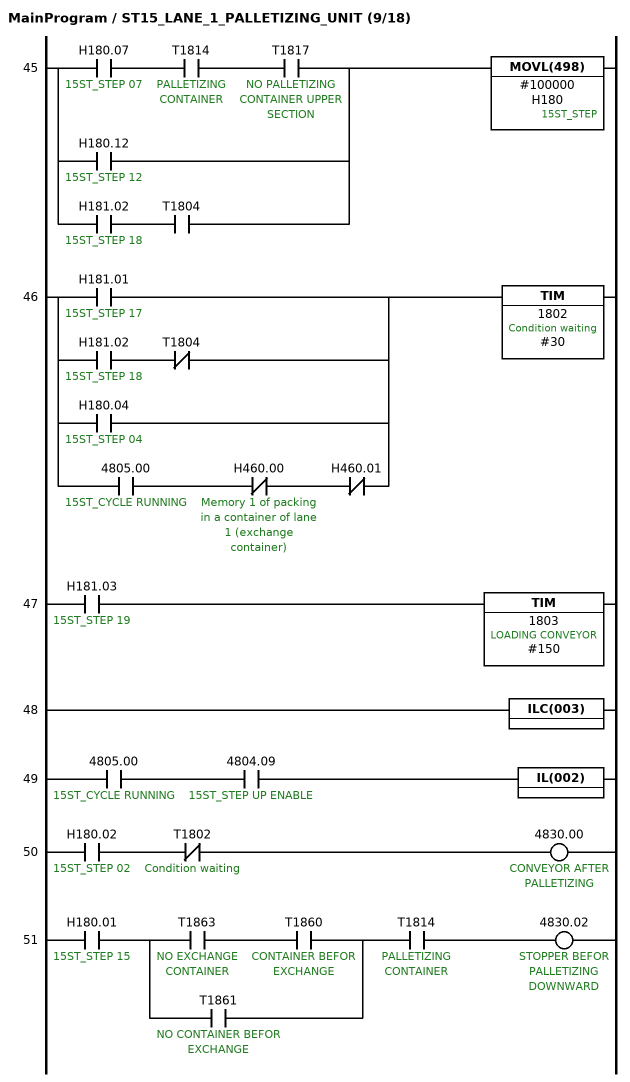
; [picture p624: MainProgram / ST15_LANE_1_PALLETIZING_UNIT, rungs 45-51]
; rung 45
LD H180.07  ; 15ST_STEP 07
AND T1814  ; PALLETIZING CONTAINER
AND T1817  ; NO PALLETIZING CONTAINER UPPER SECTION
OR H180.12  ; 15ST_STEP 12
LD H181.02  ; 15ST_STEP 18
AND T1804
ORLD
MOVL(498) #100000 H180  ; 15ST_STEP
; rung 46
LD H181.01  ; 15ST_STEP 17
LD H181.02  ; 15ST_STEP 18
ANDNOT T1804
ORLD
OR H180.04  ; 15ST_STEP 04
LD 4805.00  ; 15ST_CYCLE RUNNING
ANDNOT H460.00  ; Memory 1 of packing in a container of lane 1 (exchange container)
ANDNOT H460.01
ORLD
TIM 1802 #30  ; Condition waiting
; rung 47
LD H181.03  ; 15ST_STEP 19
TIM 1803 #150  ; LOADING CONVEYOR
; rung 48
ILC(003)
; rung 49
LD 4805.00  ; 15ST_CYCLE RUNNING
AND 4804.09  ; 15ST_STEP UP ENABLE
IL(002)
; rung 50
LD H180.02  ; 15ST_STEP 02
ANDNOT T1802  ; Condition waiting
OUT 4830.00  ; CONVEYOR AFTER PALLETIZING
; rung 51
LD H180.01  ; 15ST_STEP 15
LD T1863  ; NO EXCHANGE CONTAINER
AND T1860  ; CONTAINER BEFOR EXCHANGE
OR T1861  ; NO CONTAINER BEFOR EXCHANGE
ANDLD
AND T1814  ; PALLETIZING CONTAINER
OUT 4830.02  ; STOPPER BEFOR PALLETIZING DOWNWARD

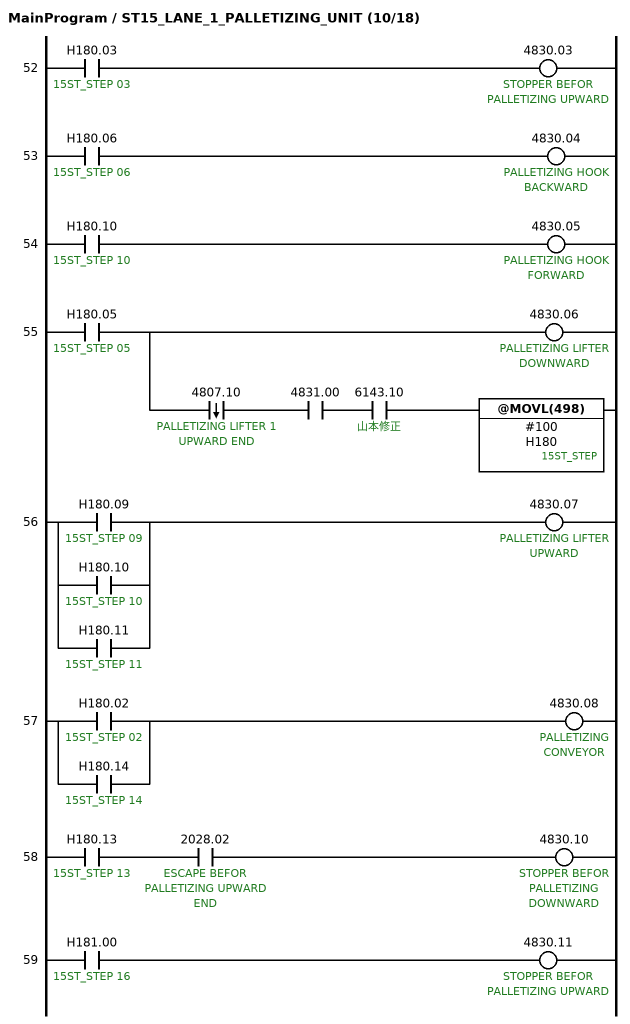
; rung 52
LD H180.03  ; 15ST_STEP 03
OUT 4830.03  ; STOPPER BEFOR PALLETIZING UPWARD
; rung 53
LD H180.06  ; 15ST_STEP 06
OUT 4830.04  ; PALLETIZING HOOK BACKWARD
; rung 54
LD H180.10  ; 15ST_STEP 10
OUT 4830.05  ; PALLETIZING HOOK FORWARD
; rung 55
LD H180.05  ; 15ST_STEP 05
OUT 4830.06  ; PALLETIZING LIFTER DOWNWARD
%AND 4807.10  ; PALLETIZING LIFTER 1 UPWARD END
AND 4831.00
AND 6143.10  ; 山本修正
@MOVL(498) #100 H180  ; 15ST_STEP
; rung 56
LD H180.09  ; 15ST_STEP 09
OR H180.10  ; 15ST_STEP 10
OR H180.11  ; 15ST_STEP 11
OUT 4830.07  ; PALLETIZING LIFTER UPWARD
; rung 57
LD H180.02  ; 15ST_STEP 02
OR H180.14  ; 15ST_STEP 14
OUT 4830.08  ; PALLETIZING CONVEYOR
; rung 58
LD H180.13  ; 15ST_STEP 13
AND 2028.02  ; ESCAPE BEFOR PALLETIZING UPWARD END
OUT 4830.10  ; STOPPER BEFOR PALLETIZING DOWNWARD
; rung 59
LD H181.00  ; 15ST_STEP 16
OUT 4830.11  ; STOPPER BEFOR PALLETIZING UPWARD

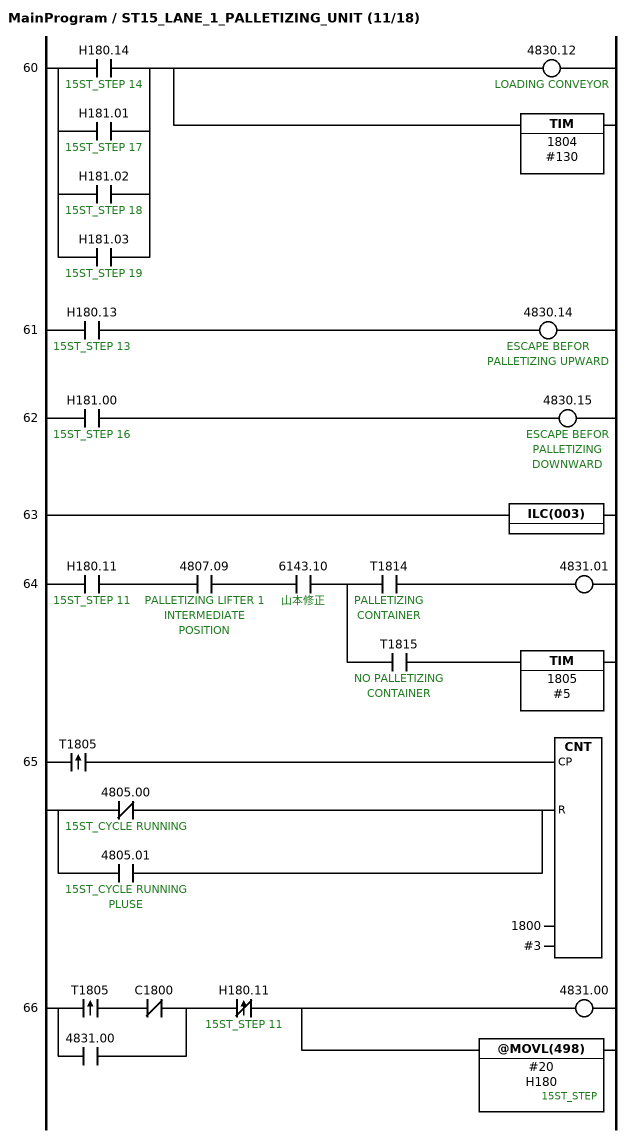
; rung 60
LD H180.14  ; 15ST_STEP 14
OR H181.01  ; 15ST_STEP 17
OR H181.02  ; 15ST_STEP 18
OR H181.03  ; 15ST_STEP 19
OUT 4830.12  ; LOADING CONVEYOR
TIM 1804 #130
; rung 61
LD H180.13  ; 15ST_STEP 13
OUT 4830.14  ; ESCAPE BEFOR PALLETIZING UPWARD
; rung 62
LD H181.00  ; 15ST_STEP 16
OUT 4830.15  ; ESCAPE BEFOR PALLETIZING DOWNWARD
; rung 63
ILC(003)
; rung 64
LD H180.11  ; 15ST_STEP 11
AND 4807.09  ; PALLETIZING LIFTER 1 INTERMEDIATE POSITION
AND 6143.10  ; 山本修正
OUT TR0
AND T1814  ; PALLETIZING CONTAINER
OUT 4831.01
LD TR0
AND T1815  ; NO PALLETIZING CONTAINER
TIM 1805 #5
; rung 65
@LD T1805
LDNOT 4805.00  ; 15ST_CYCLE RUNNING
OR 4805.01  ; 15ST_CYCLE RUNNING PLUSE
CNT 1800 #3
; rung 66
@LD T1805
ANDNOT C1800
OR 4831.00
@ANDNOT H180.11  ; 15ST_STEP 11
OUT 4831.00
@MOVL(498) #20 H180  ; 15ST_STEP

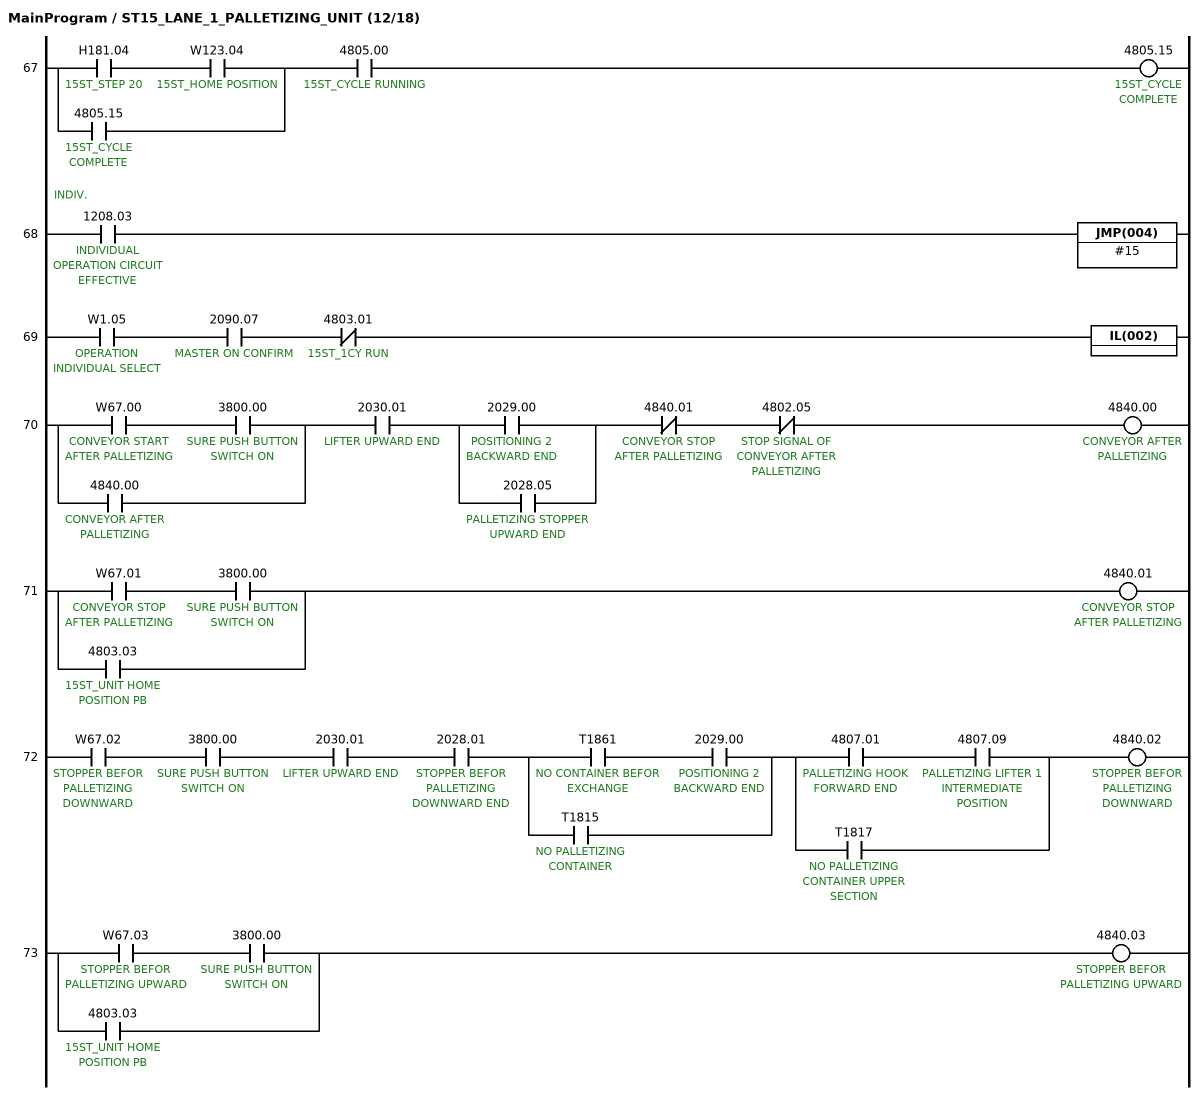
; rung 67
LD H181.04  ; 15ST_STEP 20
AND W123.04  ; 15ST_HOME POSITION
OR 4805.15  ; 15ST_CYCLE COMPLETE
AND 4805.00  ; 15ST_CYCLE RUNNING
OUT 4805.15  ; 15ST_CYCLE COMPLETE
; rung 68: INDIV.
LD 1208.03  ; INDIVIDUAL OPERATION CIRCUIT EFFECTIVE
JMP(004) #15
; rung 69
LD W1.05  ; OPERATION INDIVIDUAL SELECT
AND 2090.07  ; MASTER ON CONFIRM
ANDNOT 4803.01  ; 15ST_1CY RUN
IL(002)
; rung 70
LD W67.00  ; CONVEYOR START AFTER PALLETIZING
AND 3800.00  ; SURE PUSH BUTTON SWITCH ON
OR 4840.00  ; CONVEYOR AFTER PALLETIZING
AND 2030.01  ; LIFTER UPWARD END
LD 2029.00  ; POSITIONING 2 BACKWARD END
OR 2028.05  ; PALLETIZING STOPPER UPWARD END
ANDLD
ANDNOT 4840.01  ; CONVEYOR STOP AFTER PALLETIZING
ANDNOT 4802.05  ; STOP SIGNAL OF CONVEYOR AFTER PALLETIZING
OUT 4840.00  ; CONVEYOR AFTER PALLETIZING
; rung 71
LD W67.01  ; CONVEYOR STOP AFTER PALLETIZING
AND 3800.00  ; SURE PUSH BUTTON SWITCH ON
OR 4803.03  ; 15ST_UNIT HOME POSITION PB
OUT 4840.01  ; CONVEYOR STOP AFTER PALLETIZING
; rung 72
LD W67.02  ; STOPPER BEFOR PALLETIZING DOWNWARD
AND 3800.00  ; SURE PUSH BUTTON SWITCH ON
AND 2030.01  ; LIFTER UPWARD END
AND 2028.01  ; STOPPER BEFOR PALLETIZING DOWNWARD END
LD T1861  ; NO CONTAINER BEFOR EXCHANGE
AND 2029.00  ; POSITIONING 2 BACKWARD END
OR T1815  ; NO PALLETIZING CONTAINER
ANDLD
LD 4807.01  ; PALLETIZING HOOK FORWARD END
AND 4807.09  ; PALLETIZING LIFTER 1 INTERMEDIATE POSITION
OR T1817  ; NO PALLETIZING CONTAINER UPPER SECTION
ANDLD
OUT 4840.02  ; STOPPER BEFOR PALLETIZING DOWNWARD
; rung 73
LD W67.03  ; STOPPER BEFOR PALLETIZING UPWARD
AND 3800.00  ; SURE PUSH BUTTON SWITCH ON
OR 4803.03  ; 15ST_UNIT HOME POSITION PB
OUT 4840.03  ; STOPPER BEFOR PALLETIZING UPWARD

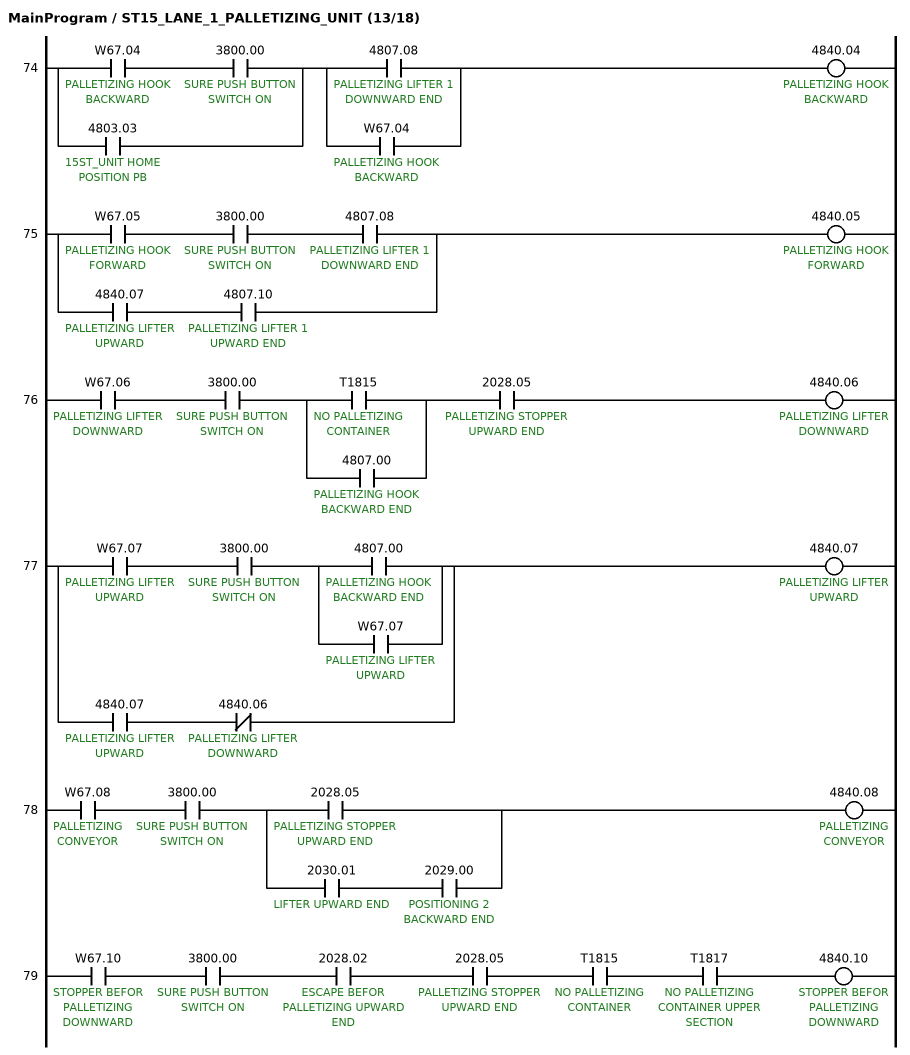
; rung 74
LD W67.04  ; PALLETIZING HOOK BACKWARD
AND 3800.00  ; SURE PUSH BUTTON SWITCH ON
OR 4803.03  ; 15ST_UNIT HOME POSITION PB
LD 4807.08  ; PALLETIZING LIFTER 1 DOWNWARD END
OR W67.04  ; PALLETIZING HOOK BACKWARD
ANDLD
OUT 4840.04  ; PALLETIZING HOOK BACKWARD
; rung 75
LD W67.05  ; PALLETIZING HOOK FORWARD
AND 3800.00  ; SURE PUSH BUTTON SWITCH ON
AND 4807.08  ; PALLETIZING LIFTER 1 DOWNWARD END
LD 4840.07  ; PALLETIZING LIFTER UPWARD
AND 4807.10  ; PALLETIZING LIFTER 1 UPWARD END
ORLD
OUT 4840.05  ; PALLETIZING HOOK FORWARD
; rung 76
LD W67.06  ; PALLETIZING LIFTER DOWNWARD
AND 3800.00  ; SURE PUSH BUTTON SWITCH ON
LD T1815  ; NO PALLETIZING CONTAINER
OR 4807.00  ; PALLETIZING HOOK BACKWARD END
ANDLD
AND 2028.05  ; PALLETIZING STOPPER UPWARD END
OUT 4840.06  ; PALLETIZING LIFTER DOWNWARD
; rung 77
LD W67.07  ; PALLETIZING LIFTER UPWARD
AND 3800.00  ; SURE PUSH BUTTON SWITCH ON
LD 4807.00  ; PALLETIZING HOOK BACKWARD END
OR W67.07  ; PALLETIZING LIFTER UPWARD
ANDLD
LD 4840.07  ; PALLETIZING LIFTER UPWARD
ANDNOT 4840.06  ; PALLETIZING LIFTER DOWNWARD
ORLD
OUT 4840.07  ; PALLETIZING LIFTER UPWARD
; rung 78
LD W67.08  ; PALLETIZING CONVEYOR
AND 3800.00  ; SURE PUSH BUTTON SWITCH ON
LD 2028.05  ; PALLETIZING STOPPER UPWARD END
LD 2030.01  ; LIFTER UPWARD END
AND 2029.00  ; POSITIONING 2 BACKWARD END
ORLD
ANDLD
OUT 4840.08  ; PALLETIZING CONVEYOR
; rung 79
LD W67.10  ; STOPPER BEFOR PALLETIZING DOWNWARD
AND 3800.00  ; SURE PUSH BUTTON SWITCH ON
AND 2028.02  ; ESCAPE BEFOR PALLETIZING UPWARD END
AND 2028.05  ; PALLETIZING STOPPER UPWARD END
AND T1815  ; NO PALLETIZING CONTAINER
AND T1817  ; NO PALLETIZING CONTAINER UPPER SECTION
OUT 4840.10  ; STOPPER BEFOR PALLETIZING DOWNWARD

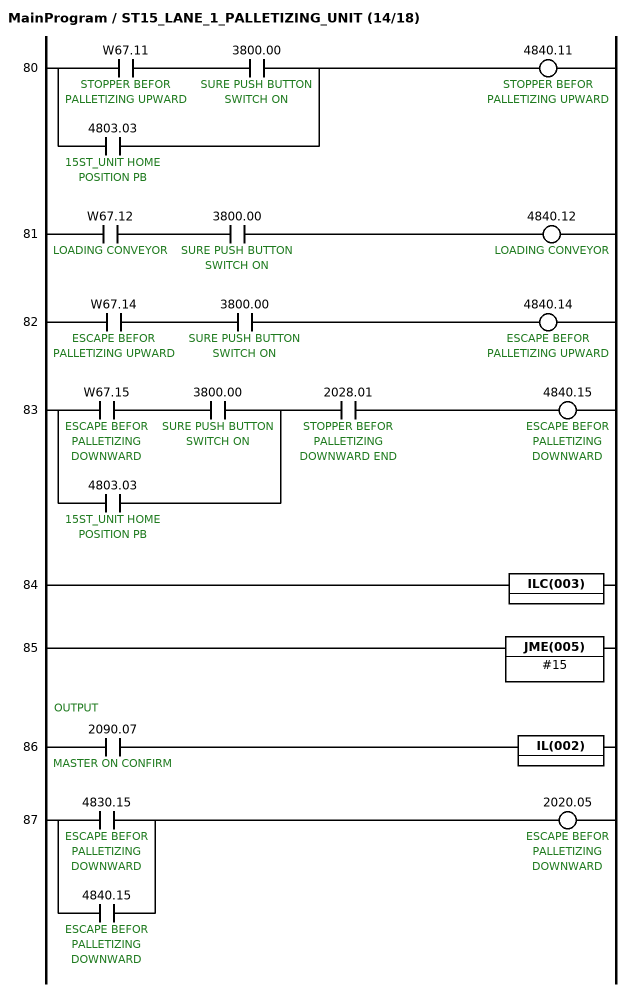
; rung 80
LD W67.11  ; STOPPER BEFOR PALLETIZING UPWARD
AND 3800.00  ; SURE PUSH BUTTON SWITCH ON
OR 4803.03  ; 15ST_UNIT HOME POSITION PB
OUT 4840.11  ; STOPPER BEFOR PALLETIZING UPWARD
; rung 81
LD W67.12  ; LOADING CONVEYOR
AND 3800.00  ; SURE PUSH BUTTON SWITCH ON
OUT 4840.12  ; LOADING CONVEYOR
; rung 82
LD W67.14  ; ESCAPE BEFOR PALLETIZING UPWARD
AND 3800.00  ; SURE PUSH BUTTON SWITCH ON
OUT 4840.14  ; ESCAPE BEFOR PALLETIZING UPWARD
; rung 83
LD W67.15  ; ESCAPE BEFOR PALLETIZING DOWNWARD
AND 3800.00  ; SURE PUSH BUTTON SWITCH ON
OR 4803.03  ; 15ST_UNIT HOME POSITION PB
AND 2028.01  ; STOPPER BEFOR PALLETIZING DOWNWARD END
OUT 4840.15  ; ESCAPE BEFOR PALLETIZING DOWNWARD
; rung 84
ILC(003)
; rung 85
JME(005) #15
; rung 86: OUTPUT
LD 2090.07  ; MASTER ON CONFIRM
IL(002)
; rung 87
LD 4830.15  ; ESCAPE BEFOR PALLETIZING DOWNWARD
OR 4840.15  ; ESCAPE BEFOR PALLETIZING DOWNWARD
OUT 2020.05  ; ESCAPE BEFOR PALLETIZING DOWNWARD

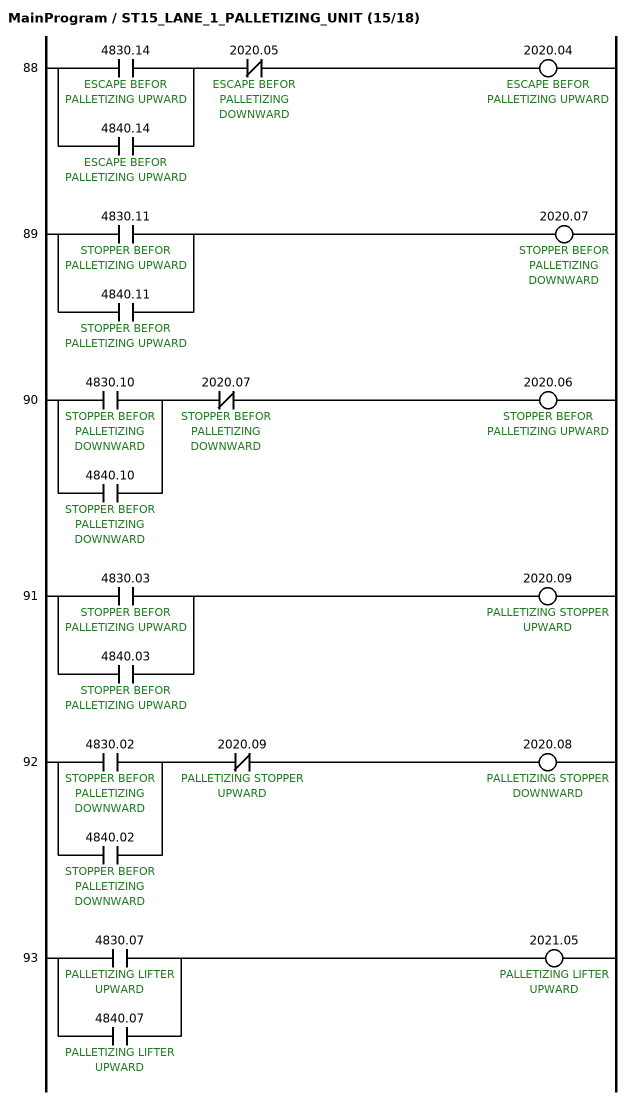
; rung 88
LD 4830.14  ; ESCAPE BEFOR PALLETIZING UPWARD
OR 4840.14  ; ESCAPE BEFOR PALLETIZING UPWARD
ANDNOT 2020.05  ; ESCAPE BEFOR PALLETIZING DOWNWARD
OUT 2020.04  ; ESCAPE BEFOR PALLETIZING UPWARD
; rung 89
LD 4830.11  ; STOPPER BEFOR PALLETIZING UPWARD
OR 4840.11  ; STOPPER BEFOR PALLETIZING UPWARD
OUT 2020.07  ; STOPPER BEFOR PALLETIZING DOWNWARD
; rung 90
LD 4830.10  ; STOPPER BEFOR PALLETIZING DOWNWARD
OR 4840.10  ; STOPPER BEFOR PALLETIZING DOWNWARD
ANDNOT 2020.07  ; STOPPER BEFOR PALLETIZING DOWNWARD
OUT 2020.06  ; STOPPER BEFOR PALLETIZING UPWARD
; rung 91
LD 4830.03  ; STOPPER BEFOR PALLETIZING UPWARD
OR 4840.03  ; STOPPER BEFOR PALLETIZING UPWARD
OUT 2020.09  ; PALLETIZING STOPPER UPWARD
; rung 92
LD 4830.02  ; STOPPER BEFOR PALLETIZING DOWNWARD
OR 4840.02  ; STOPPER BEFOR PALLETIZING DOWNWARD
ANDNOT 2020.09  ; PALLETIZING STOPPER UPWARD
OUT 2020.08  ; PALLETIZING STOPPER DOWNWARD
; rung 93
LD 4830.07  ; PALLETIZING LIFTER UPWARD
OR 4840.07  ; PALLETIZING LIFTER UPWARD
OUT 2021.05  ; PALLETIZING LIFTER UPWARD

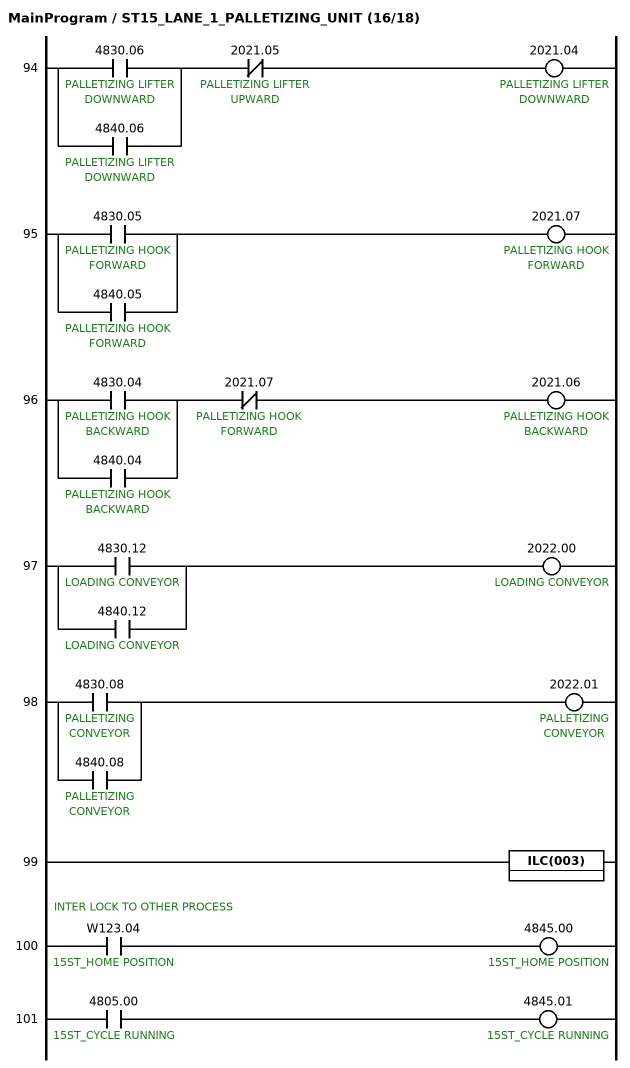
; rung 94
LD 4830.06  ; PALLETIZING LIFTER DOWNWARD
OR 4840.06  ; PALLETIZING LIFTER DOWNWARD
ANDNOT 2021.05  ; PALLETIZING LIFTER UPWARD
OUT 2021.04  ; PALLETIZING LIFTER DOWNWARD
; rung 95
LD 4830.05  ; PALLETIZING HOOK FORWARD
OR 4840.05  ; PALLETIZING HOOK FORWARD
OUT 2021.07  ; PALLETIZING HOOK FORWARD
; rung 96
LD 4830.04  ; PALLETIZING HOOK BACKWARD
OR 4840.04  ; PALLETIZING HOOK BACKWARD
ANDNOT 2021.07  ; PALLETIZING HOOK FORWARD
OUT 2021.06  ; PALLETIZING HOOK BACKWARD
; rung 97
LD 4830.12  ; LOADING CONVEYOR
OR 4840.12  ; LOADING CONVEYOR
OUT 2022.00  ; LOADING CONVEYOR
; rung 98
LD 4830.08  ; PALLETIZING CONVEYOR
OR 4840.08  ; PALLETIZING CONVEYOR
OUT 2022.01  ; PALLETIZING CONVEYOR
; rung 99
ILC(003)
; rung 100: INTER LOCK TO OTHER PROCESS
LD W123.04  ; 15ST_HOME POSITION
OUT 4845.00  ; 15ST_HOME POSITION
; rung 101
LD 4805.00  ; 15ST_CYCLE RUNNING
OUT 4845.01  ; 15ST_CYCLE RUNNING

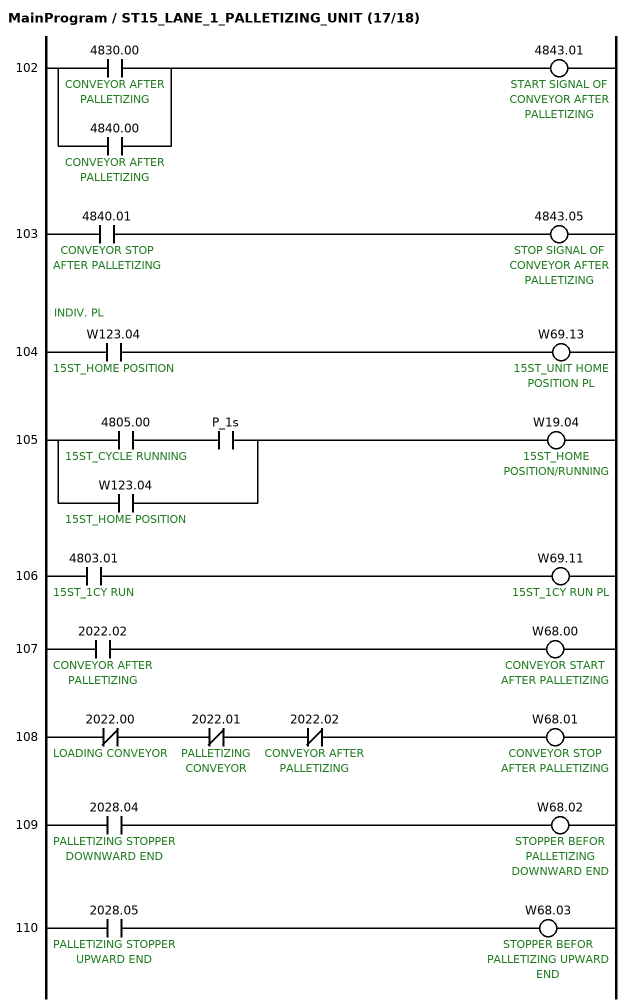
; rung 102
LD 4830.00  ; CONVEYOR AFTER PALLETIZING
OR 4840.00  ; CONVEYOR AFTER PALLETIZING
OUT 4843.01  ; START SIGNAL OF CONVEYOR AFTER PALLETIZING
; rung 103
LD 4840.01  ; CONVEYOR STOP AFTER PALLETIZING
OUT 4843.05  ; STOP SIGNAL OF CONVEYOR AFTER PALLETIZING
; rung 104: INDIV. PL
LD W123.04  ; 15ST_HOME POSITION
OUT W69.13  ; 15ST_UNIT HOME POSITION PL
; rung 105
LD 4805.00  ; 15ST_CYCLE RUNNING
AND P_1s
OR W123.04  ; 15ST_HOME POSITION
OUT W19.04  ; 15ST_HOME POSITION/RUNNING
; rung 106
LD 4803.01  ; 15ST_1CY RUN
OUT W69.11  ; 15ST_1CY RUN PL
; rung 107
LD 2022.02  ; CONVEYOR AFTER PALLETIZING
OUT W68.00  ; CONVEYOR START AFTER PALLETIZING
; rung 108
LDNOT 2022.00  ; LOADING CONVEYOR
ANDNOT 2022.01  ; PALLETIZING CONVEYOR
ANDNOT 2022.02  ; CONVEYOR AFTER PALLETIZING
OUT W68.01  ; CONVEYOR STOP AFTER PALLETIZING
; rung 109
LD 2028.04  ; PALLETIZING STOPPER DOWNWARD END
OUT W68.02  ; STOPPER BEFOR PALLETIZING DOWNWARD END
; rung 110
LD 2028.05  ; PALLETIZING STOPPER UPWARD END
OUT W68.03  ; STOPPER BEFOR PALLETIZING UPWARD END

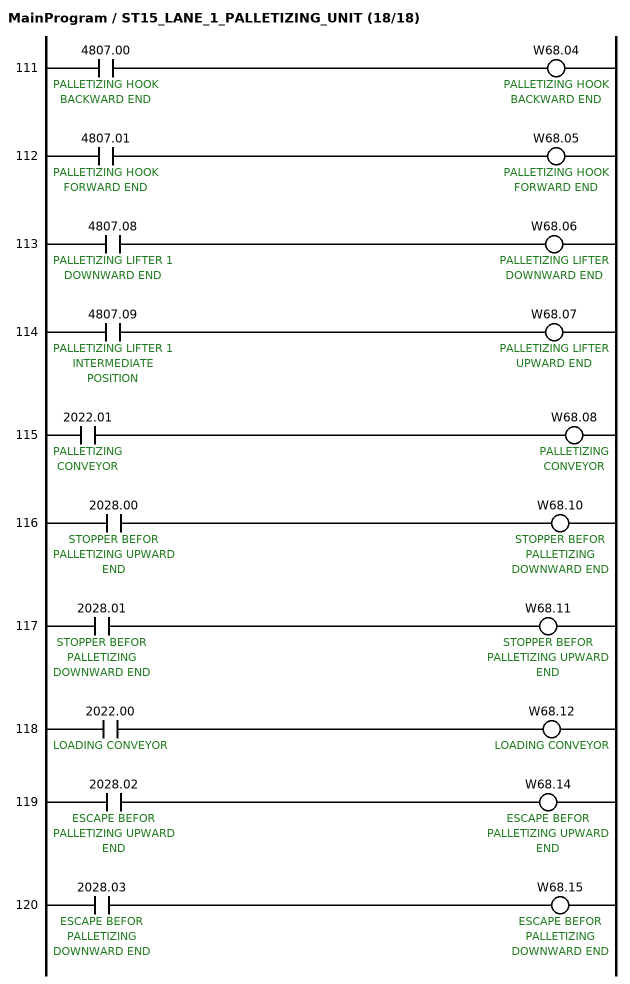
; rung 111
LD 4807.00  ; PALLETIZING HOOK BACKWARD END
OUT W68.04  ; PALLETIZING HOOK BACKWARD END
; rung 112
LD 4807.01  ; PALLETIZING HOOK FORWARD END
OUT W68.05  ; PALLETIZING HOOK FORWARD END
; rung 113
LD 4807.08  ; PALLETIZING LIFTER 1 DOWNWARD END
OUT W68.06  ; PALLETIZING LIFTER DOWNWARD END
; rung 114
LD 4807.09  ; PALLETIZING LIFTER 1 INTERMEDIATE POSITION
OUT W68.07  ; PALLETIZING LIFTER UPWARD END
; rung 115
LD 2022.01  ; PALLETIZING CONVEYOR
OUT W68.08  ; PALLETIZING CONVEYOR
; rung 116
LD 2028.00  ; STOPPER BEFOR PALLETIZING UPWARD END
OUT W68.10  ; STOPPER BEFOR PALLETIZING DOWNWARD END
; rung 117
LD 2028.01  ; STOPPER BEFOR PALLETIZING DOWNWARD END
OUT W68.11  ; STOPPER BEFOR PALLETIZING UPWARD END
; rung 118
LD 2022.00  ; LOADING CONVEYOR
OUT W68.12  ; LOADING CONVEYOR
; rung 119
LD 2028.02  ; ESCAPE BEFOR PALLETIZING UPWARD END
OUT W68.14  ; ESCAPE BEFOR PALLETIZING UPWARD END
; rung 120
LD 2028.03  ; ESCAPE BEFOR PALLETIZING DOWNWARD END
OUT W68.15  ; ESCAPE BEFOR PALLETIZING DOWNWARD END
; rung 121: CONDITION PL

### Section ST16_LANE_1_SUPPLYING_UNIT

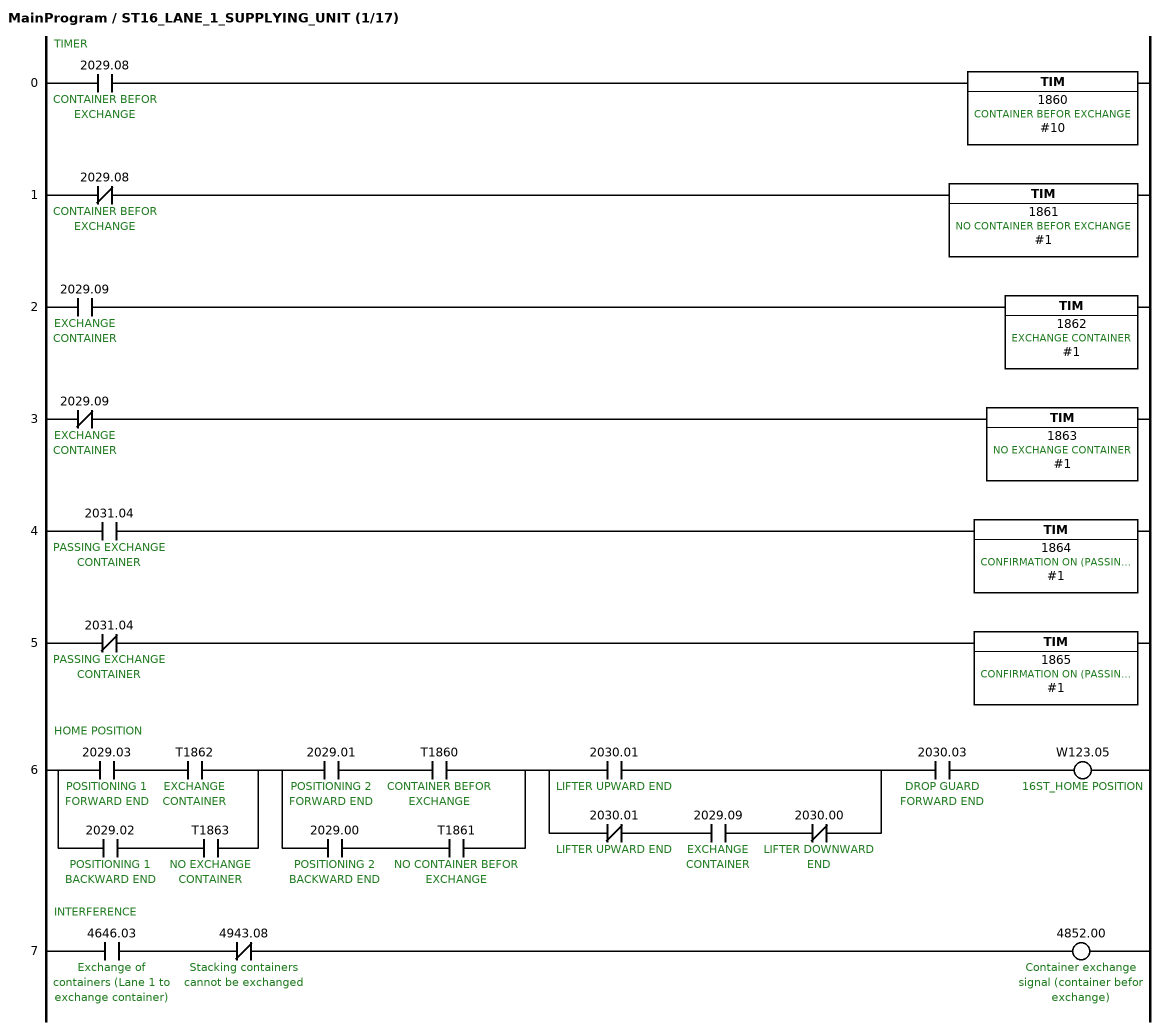
; rung 0: TIMER
LD 2029.08  ; CONTAINER BEFOR EXCHANGE
TIM 1860 #10  ; CONTAINER BEFOR EXCHANGE
; rung 1
LDNOT 2029.08  ; CONTAINER BEFOR EXCHANGE
TIM 1861 #1  ; NO CONTAINER BEFOR EXCHANGE
; rung 2
LD 2029.09  ; EXCHANGE CONTAINER
TIM 1862 #1  ; EXCHANGE CONTAINER
; rung 3
LDNOT 2029.09  ; EXCHANGE CONTAINER
TIM 1863 #1  ; NO EXCHANGE CONTAINER
; rung 4
LD 2031.04  ; PASSING EXCHANGE CONTAINER
TIM 1864 #1  ; CONFIRMATION ON (PASSING EXCHANGE CONTAINER)
; rung 5
LDNOT 2031.04  ; PASSING EXCHANGE CONTAINER
TIM 1865 #1  ; CONFIRMATION ON (PASSING EXCHANGE CONTAINER)
; rung 6: HOME POSITION
LD 2029.03  ; POSITIONING 1 FORWARD END
AND T1862  ; EXCHANGE CONTAINER
LD 2029.02  ; POSITIONING 1 BACKWARD END
AND T1863  ; NO EXCHANGE CONTAINER
ORLD
LD 2029.01  ; POSITIONING 2 FORWARD END
AND T1860  ; CONTAINER BEFOR EXCHANGE
LD 2029.00  ; POSITIONING 2 BACKWARD END
AND T1861  ; NO CONTAINER BEFOR EXCHANGE
ORLD
ANDLD
LD 2030.01  ; LIFTER UPWARD END
LDNOT 2030.01  ; LIFTER UPWARD END
AND 2029.09  ; EXCHANGE CONTAINER
ANDNOT 2030.00  ; LIFTER DOWNWARD END
ORLD
ANDLD
AND 2030.03  ; DROP GUARD FORWARD END
OUT W123.05  ; 16ST_HOME POSITION
; rung 7: INTERFERENCE
LD 4646.03  ; Exchange of containers (Lane 1 to exchange container)
ANDNOT 4943.08  ; Stacking containers cannot be exchanged
OUT 4852.00  ; Container exchange signal (container befor exchange)

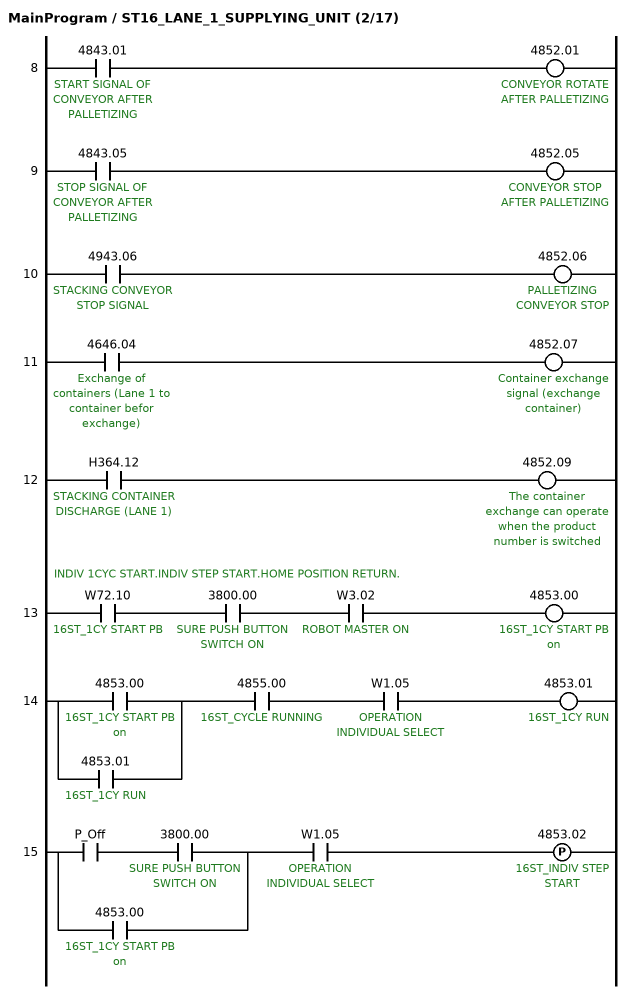
; rung 8
LD 4843.01  ; START SIGNAL OF CONVEYOR AFTER PALLETIZING
OUT 4852.01  ; CONVEYOR ROTATE AFTER PALLETIZING
; rung 9
LD 4843.05  ; STOP SIGNAL OF CONVEYOR AFTER PALLETIZING
OUT 4852.05  ; CONVEYOR STOP AFTER PALLETIZING
; rung 10
LD 4943.06  ; STACKING CONVEYOR STOP SIGNAL
OUT 4852.06  ; PALLETIZING CONVEYOR STOP
; rung 11
LD 4646.04  ; Exchange of containers (Lane 1 to container befor exchange)
OUT 4852.07  ; Container exchange signal (exchange container)
; rung 12
LD H364.12  ; STACKING CONTAINER DISCHARGE (LANE 1)
OUT 4852.09  ; The container exchange can operate when the product number is switched
; rung 13: INDIV 1CYC START.INDIV STEP START.HOME POSITION RETURN.
LD W72.10  ; 16ST_1CY START PB
AND 3800.00  ; SURE PUSH BUTTON SWITCH ON
AND W3.02  ; ROBOT MASTER ON
OUT 4853.00  ; 16ST_1CY START PB on
; rung 14
LD 4853.00  ; 16ST_1CY START PB on
OR 4853.01  ; 16ST_1CY RUN
AND 4855.00  ; 16ST_CYCLE RUNNING
AND W1.05  ; OPERATION INDIVIDUAL SELECT
OUT 4853.01  ; 16ST_1CY RUN
; rung 15
LD P_Off
AND 3800.00  ; SURE PUSH BUTTON SWITCH ON
OR 4853.00  ; 16ST_1CY START PB on
AND W1.05  ; OPERATION INDIVIDUAL SELECT
DIFU(013) 4853.02  ; 16ST_INDIV STEP START

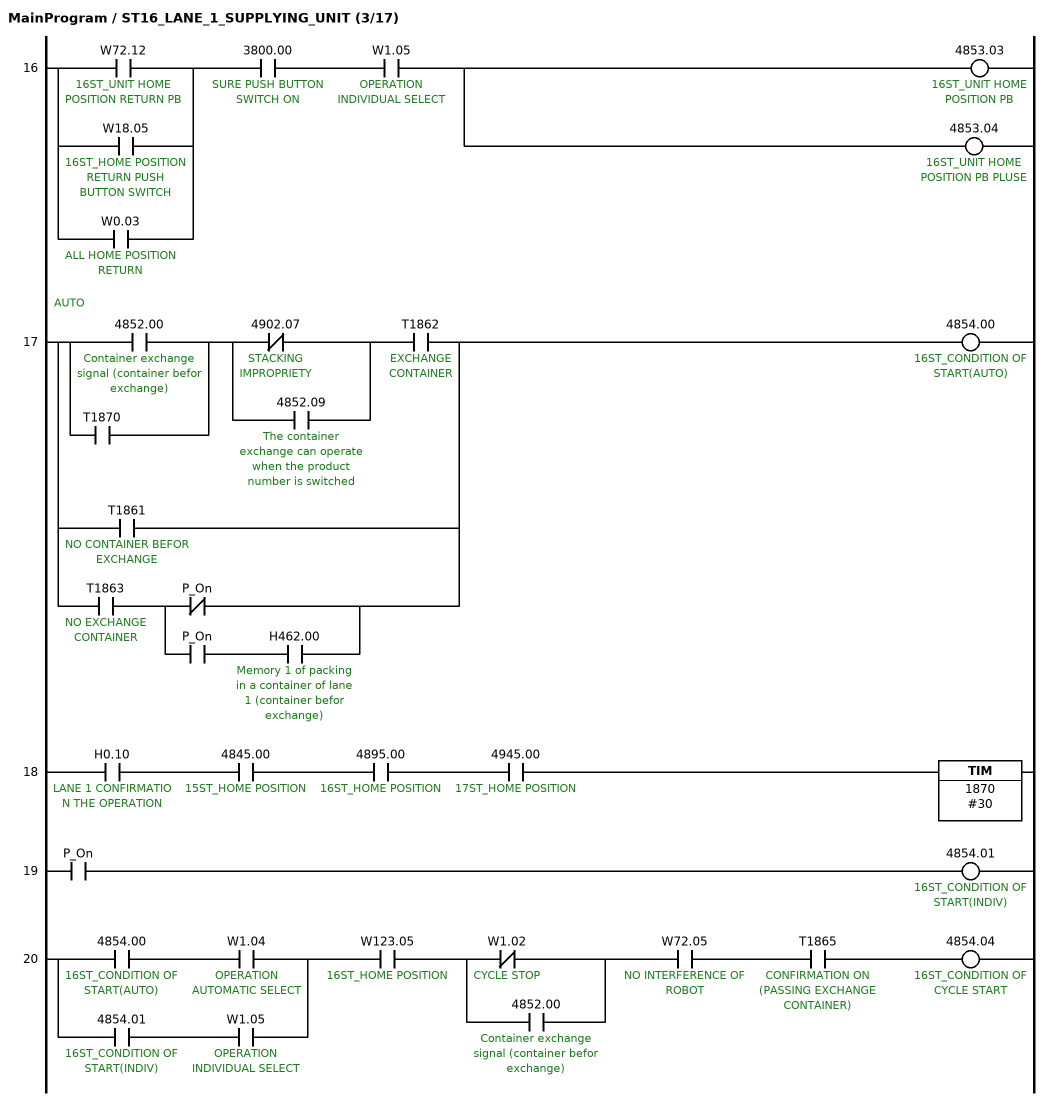
; rung 16
LD W72.12  ; 16ST_UNIT HOME POSITION RETURN PB
OR W18.05  ; 16ST_HOME POSITION RETURN PUSH BUTTON SWITCH
OR W0.03  ; ALL HOME POSITION RETURN
AND 3800.00  ; SURE PUSH BUTTON SWITCH ON
AND W1.05  ; OPERATION INDIVIDUAL SELECT
OUT 4853.03  ; 16ST_UNIT HOME POSITION PB
OUT 4853.04  ; 16ST_UNIT HOME POSITION PB PLUSE
; rung 17: AUTO
LD 4852.00  ; Container exchange signal (container befor exchange)
OR T1870
LDNOT 4902.07  ; STACKING IMPROPRIETY
OR 4852.09  ; The container exchange can operate when the product number is switched
ANDLD
AND T1862  ; EXCHANGE CONTAINER
OR T1861  ; NO CONTAINER BEFOR EXCHANGE
LD T1863  ; NO EXCHANGE CONTAINER
LDNOT P_On
LD P_On
AND H462.00  ; Memory 1 of packing in a container of lane 1 (container befor exchange)
ORLD
ANDLD
ORLD
OUT 4854.00  ; 16ST_CONDITION OF START(AUTO)
; rung 18
LD H0.10  ; LANE 1 CONFIRMATION THE OPERATION
AND 4845.00  ; 15ST_HOME POSITION
AND 4895.00  ; 16ST_HOME POSITION
AND 4945.00  ; 17ST_HOME POSITION
TIM 1870 #30
; rung 19
LD P_On
OUT 4854.01  ; 16ST_CONDITION OF START(INDIV)
; rung 20
LD 4854.00  ; 16ST_CONDITION OF START(AUTO)
AND W1.04  ; OPERATION AUTOMATIC SELECT
LD 4854.01  ; 16ST_CONDITION OF START(INDIV)
AND W1.05  ; OPERATION INDIVIDUAL SELECT
ORLD
AND W123.05  ; 16ST_HOME POSITION
LDNOT W1.02  ; CYCLE STOP
OR 4852.00  ; Container exchange signal (container befor exchange)
ANDLD
AND W72.05  ; NO INTERFERENCE OF ROBOT
AND T1865  ; CONFIRMATION ON (PASSING EXCHANGE CONTAINER)
OUT 4854.04  ; 16ST_CONDITION OF CYCLE START

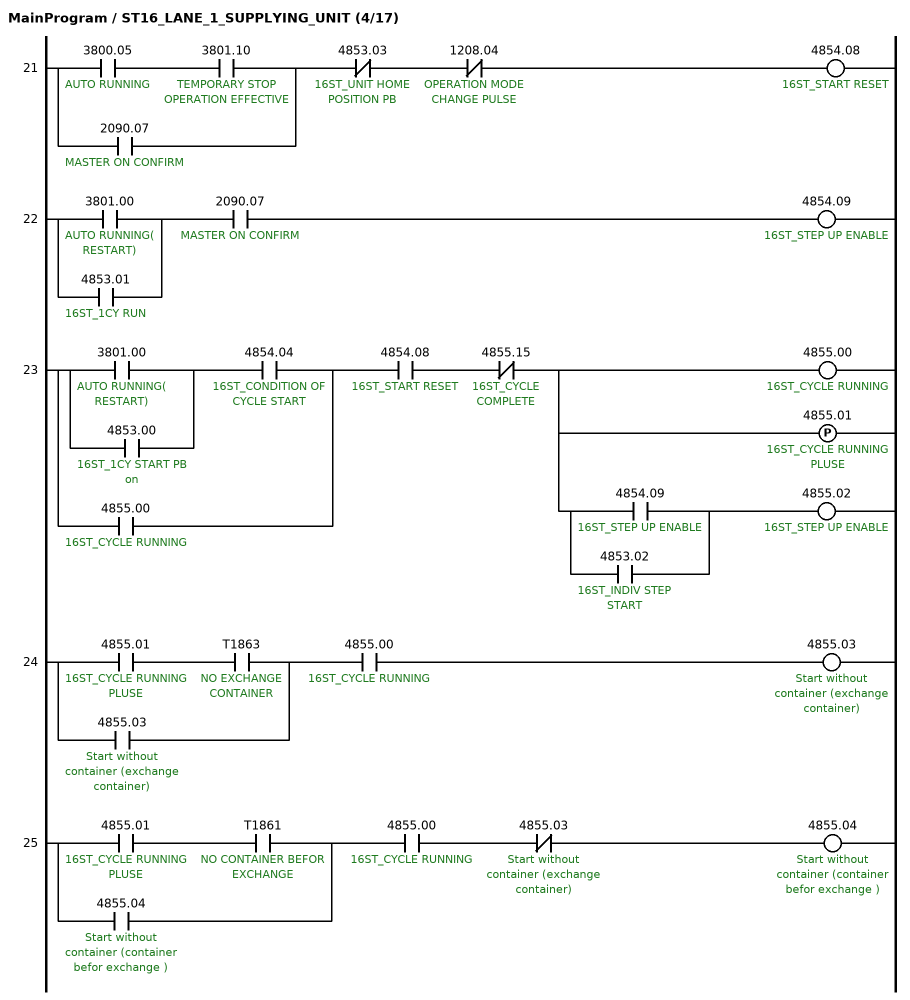
; rung 21
LD 3800.05  ; AUTO RUNNING
AND 3801.10  ; TEMPORARY STOP OPERATION EFFECTIVE
OR 2090.07  ; MASTER ON CONFIRM
ANDNOT 4853.03  ; 16ST_UNIT HOME POSITION PB
ANDNOT 1208.04  ; OPERATION MODE CHANGE PULSE
OUT 4854.08  ; 16ST_START RESET
; rung 22
LD 3801.00  ; AUTO RUNNING(RESTART)
OR 4853.01  ; 16ST_1CY RUN
AND 2090.07  ; MASTER ON CONFIRM
OUT 4854.09  ; 16ST_STEP UP ENABLE
; rung 23
LD 3801.00  ; AUTO RUNNING(RESTART)
OR 4853.00  ; 16ST_1CY START PB on
AND 4854.04  ; 16ST_CONDITION OF CYCLE START
OR 4855.00  ; 16ST_CYCLE RUNNING
AND 4854.08  ; 16ST_START RESET
ANDNOT 4855.15  ; 16ST_CYCLE COMPLETE
OUT 4855.00  ; 16ST_CYCLE RUNNING
DIFU(013) 4855.01  ; 16ST_CYCLE RUNNING PLUSE
LD 4854.09  ; 16ST_STEP UP ENABLE
OR 4853.02  ; 16ST_INDIV STEP START
ANDLD
OUT 4855.02  ; 16ST_STEP UP ENABLE
; rung 24
LD 4855.01  ; 16ST_CYCLE RUNNING PLUSE
AND T1863  ; NO EXCHANGE CONTAINER
OR 4855.03  ; Start without container (exchange container)
AND 4855.00  ; 16ST_CYCLE RUNNING
OUT 4855.03  ; Start without container (exchange container)
; rung 25
LD 4855.01  ; 16ST_CYCLE RUNNING PLUSE
AND T1861  ; NO CONTAINER BEFOR EXCHANGE
OR 4855.04  ; Start without container (container befor exchange )
AND 4855.00  ; 16ST_CYCLE RUNNING
ANDNOT 4855.03  ; Start without container (exchange container)
OUT 4855.04  ; Start without container (container befor exchange )

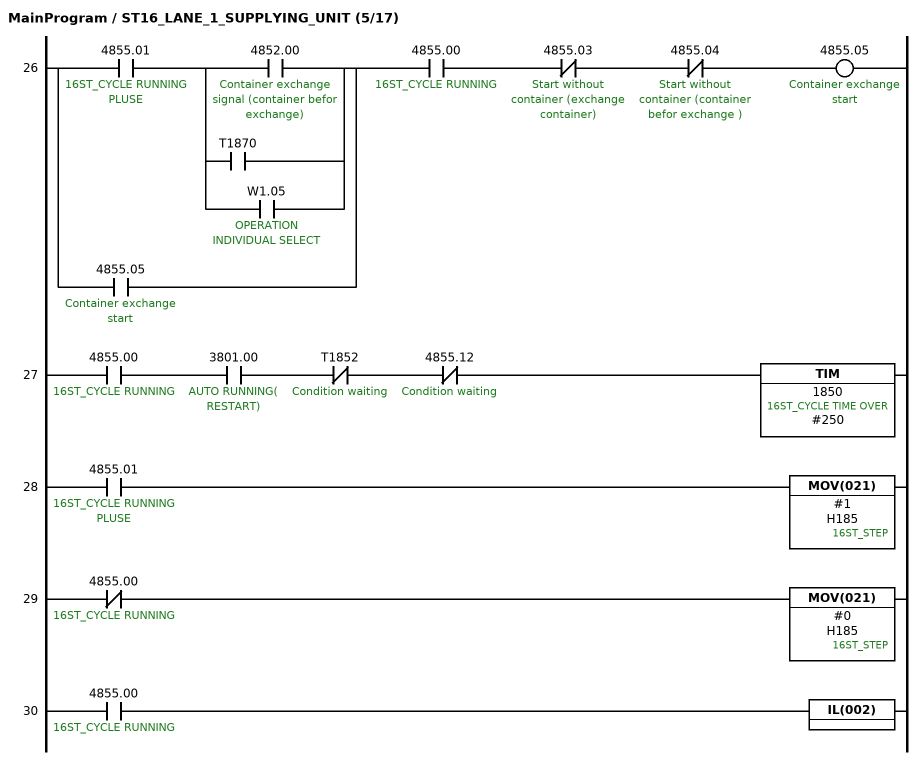
; rung 26
LD 4855.01  ; 16ST_CYCLE RUNNING PLUSE
LD 4852.00  ; Container exchange signal (container befor exchange)
OR T1870
OR W1.05  ; OPERATION INDIVIDUAL SELECT
ANDLD
OR 4855.05  ; Container exchange start
AND 4855.00  ; 16ST_CYCLE RUNNING
ANDNOT 4855.03  ; Start without container (exchange container)
ANDNOT 4855.04  ; Start without container (container befor exchange )
OUT 4855.05  ; Container exchange start
; rung 27
LD 4855.00  ; 16ST_CYCLE RUNNING
AND 3801.00  ; AUTO RUNNING(RESTART)
ANDNOT T1852  ; Condition waiting
ANDNOT 4855.12  ; Condition waiting
TIM 1850 #250  ; 16ST_CYCLE TIME OVER
; rung 28
LD 4855.01  ; 16ST_CYCLE RUNNING PLUSE
MOV(021) #1 H185  ; 16ST_STEP
; rung 29
LDNOT 4855.00  ; 16ST_CYCLE RUNNING
MOV(021) #0 H185  ; 16ST_STEP
; rung 30
LD 4855.00  ; 16ST_CYCLE RUNNING
IL(002)

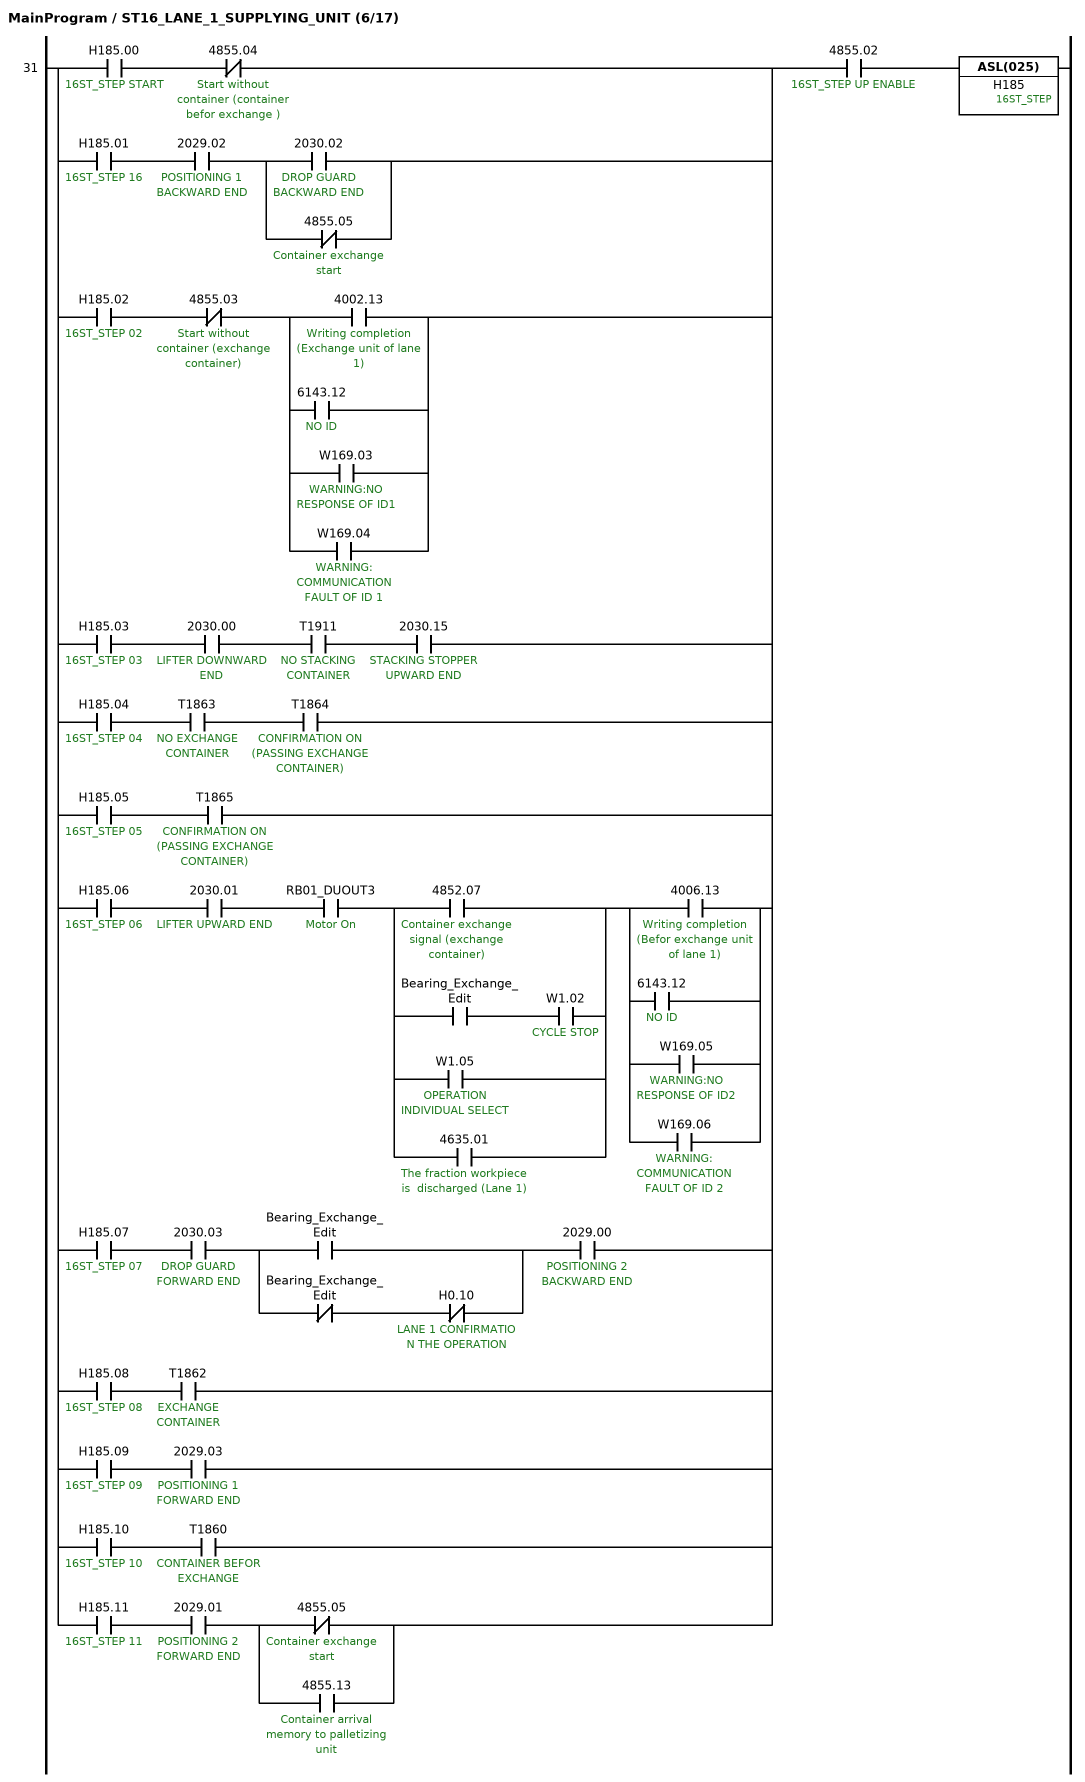
; rung 31
LD H185.00  ; 16ST_STEP START
ANDNOT 4855.04  ; Start without container (container befor exchange )
LD H185.01  ; 16ST_STEP 16
AND 2029.02  ; POSITIONING 1 BACKWARD END
LD 2030.02  ; DROP GUARD BACKWARD END
ORNOT 4855.05  ; Container exchange start
ANDLD
ORLD
LD H185.02  ; 16ST_STEP 02
ANDNOT 4855.03  ; Start without container (exchange container)
LD 4002.13  ; Writing completion (Exchange unit of lane 1)
OR 6143.12  ; NO ID
OR W169.03  ; WARNING:NO RESPONSE OF ID1
OR W169.04  ; WARNING:COMMUNICATION FAULT OF ID 1
ANDLD
ORLD
LD H185.03  ; 16ST_STEP 03
AND 2030.00  ; LIFTER DOWNWARD END
AND T1911  ; NO STACKING CONTAINER
AND 2030.15  ; STACKING STOPPER UPWARD END
ORLD
LD H185.04  ; 16ST_STEP 04
AND T1863  ; NO EXCHANGE CONTAINER
AND T1864  ; CONFIRMATION ON (PASSING EXCHANGE CONTAINER)
ORLD
LD H185.05  ; 16ST_STEP 05
AND T1865  ; CONFIRMATION ON (PASSING EXCHANGE CONTAINER)
ORLD
LD H185.06  ; 16ST_STEP 06
AND 2030.01  ; LIFTER UPWARD END
AND RB01_DUOUT3  ; Motor On
LD 4852.07  ; Container exchange signal (exchange container)
LD Bearing_Exchange_Edit
AND W1.02  ; CYCLE STOP
ORLD
OR W1.05  ; OPERATION INDIVIDUAL SELECT
OR 4635.01  ; The fraction workpiece is  discharged (Lane 1)
ANDLD
LD 4006.13  ; Writing completion (Befor exchange unit of lane 1)
OR 6143.12  ; NO ID
OR W169.05  ; WARNING:NO RESPONSE OF ID2
OR W169.06  ; WARNING:COMMUNICATION FAULT OF ID 2
ANDLD
ORLD
LD H185.07  ; 16ST_STEP 07
AND 2030.03  ; DROP GUARD FORWARD END
LD Bearing_Exchange_Edit
LDNOT Bearing_Exchange_Edit
ANDNOT H0.10  ; LANE 1 CONFIRMATION THE OPERATION
ORLD
ANDLD
AND 2029.00  ; POSITIONING 2 BACKWARD END
ORLD
LD H185.08  ; 16ST_STEP 08
AND T1862  ; EXCHANGE CONTAINER
ORLD
LD H185.09  ; 16ST_STEP 09
AND 2029.03  ; POSITIONING 1 FORWARD END
ORLD
LD H185.10  ; 16ST_STEP 10
AND T1860  ; CONTAINER BEFOR EXCHANGE
ORLD
LD H185.11  ; 16ST_STEP 11
AND 2029.01  ; POSITIONING 2 FORWARD END
LDNOT 4855.05  ; Container exchange start
OR 4855.13  ; Container arrival memory to palletizing unit
ANDLD
ORLD
AND 4855.02  ; 16ST_STEP UP ENABLE
ASL(025) H185  ; 16ST_STEP

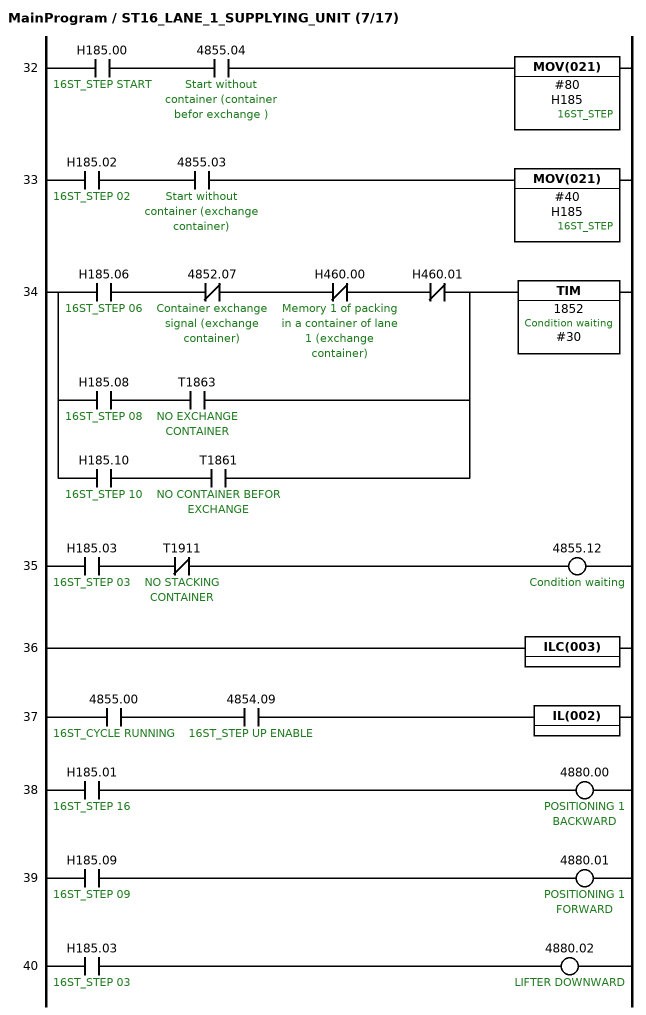
; rung 32
LD H185.00  ; 16ST_STEP START
AND 4855.04  ; Start without container (container befor exchange )
MOV(021) #80 H185  ; 16ST_STEP
; rung 33
LD H185.02  ; 16ST_STEP 02
AND 4855.03  ; Start without container (exchange container)
MOV(021) #40 H185  ; 16ST_STEP
; rung 34
LD H185.06  ; 16ST_STEP 06
ANDNOT 4852.07  ; Container exchange signal (exchange container)
ANDNOT H460.00  ; Memory 1 of packing in a container of lane 1 (exchange container)
ANDNOT H460.01
LD H185.08  ; 16ST_STEP 08
AND T1863  ; NO EXCHANGE CONTAINER
ORLD
LD H185.10  ; 16ST_STEP 10
AND T1861  ; NO CONTAINER BEFOR EXCHANGE
ORLD
TIM 1852 #30  ; Condition waiting
; rung 35
LD H185.03  ; 16ST_STEP 03
ANDNOT T1911  ; NO STACKING CONTAINER
OUT 4855.12  ; Condition waiting
; rung 36
ILC(003)
; rung 37
LD 4855.00  ; 16ST_CYCLE RUNNING
AND 4854.09  ; 16ST_STEP UP ENABLE
IL(002)
; rung 38
LD H185.01  ; 16ST_STEP 16
OUT 4880.00  ; POSITIONING 1 BACKWARD
; rung 39
LD H185.09  ; 16ST_STEP 09
OUT 4880.01  ; POSITIONING 1 FORWARD
; rung 40
LD H185.03  ; 16ST_STEP 03
OUT 4880.02  ; LIFTER DOWNWARD

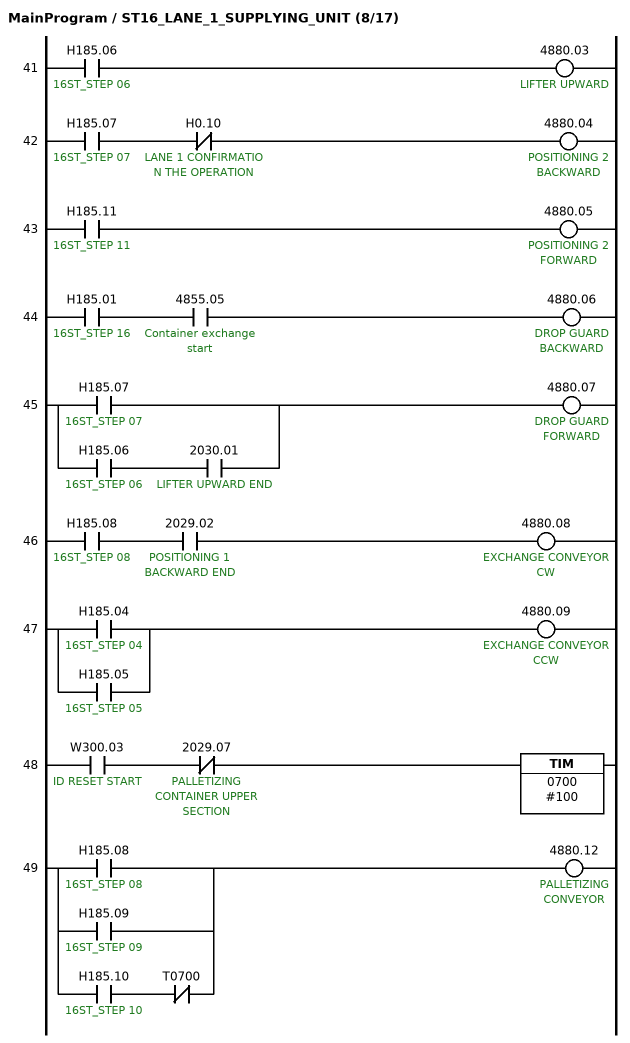
; rung 41
LD H185.06  ; 16ST_STEP 06
OUT 4880.03  ; LIFTER UPWARD
; rung 42
LD H185.07  ; 16ST_STEP 07
ANDNOT H0.10  ; LANE 1 CONFIRMATION THE OPERATION
OUT 4880.04  ; POSITIONING 2 BACKWARD
; rung 43
LD H185.11  ; 16ST_STEP 11
OUT 4880.05  ; POSITIONING 2 FORWARD
; rung 44
LD H185.01  ; 16ST_STEP 16
AND 4855.05  ; Container exchange start
OUT 4880.06  ; DROP GUARD BACKWARD
; rung 45
LD H185.07  ; 16ST_STEP 07
LD H185.06  ; 16ST_STEP 06
AND 2030.01  ; LIFTER UPWARD END
ORLD
OUT 4880.07  ; DROP GUARD FORWARD
; rung 46
LD H185.08  ; 16ST_STEP 08
AND 2029.02  ; POSITIONING 1 BACKWARD END
OUT 4880.08  ; EXCHANGE CONVEYOR CW
; rung 47
LD H185.04  ; 16ST_STEP 04
OR H185.05  ; 16ST_STEP 05
OUT 4880.09  ; EXCHANGE CONVEYOR CCW
; rung 48
LD W300.03  ; ID RESET START
ANDNOT 2029.07  ; PALLETIZING CONTAINER UPPER SECTION
TIM 0700 #100
; rung 49
LD H185.08  ; 16ST_STEP 08
OR H185.09  ; 16ST_STEP 09
LD H185.10  ; 16ST_STEP 10
ANDNOT T0700
ORLD
OUT 4880.12  ; PALLETIZING CONVEYOR

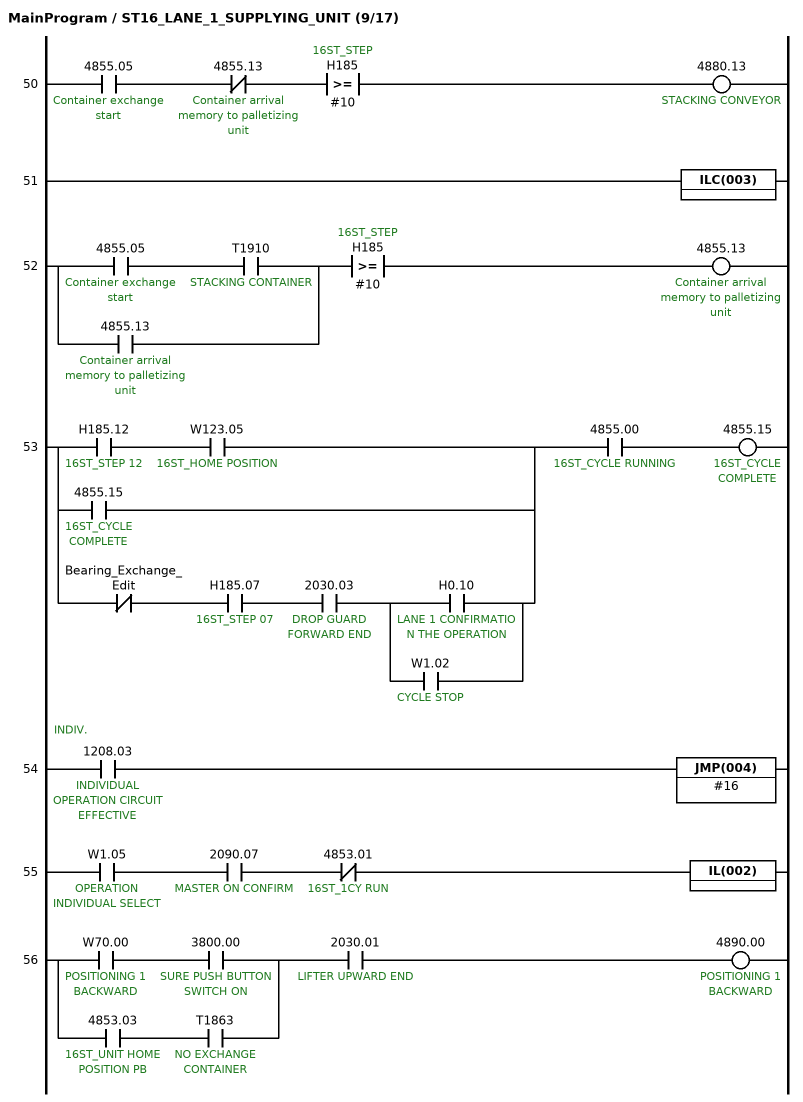
; rung 50
LD 4855.05  ; Container exchange start
ANDNOT 4855.13  ; Container arrival memory to palletizing unit
AND>=(325) H185 #10  ; 16ST_STEP
OUT 4880.13  ; STACKING CONVEYOR
; rung 51
ILC(003)
; rung 52
LD 4855.05  ; Container exchange start
AND T1910  ; STACKING CONTAINER
OR 4855.13  ; Container arrival memory to palletizing unit
AND>=(325) H185 #10  ; 16ST_STEP
OUT 4855.13  ; Container arrival memory to palletizing unit
; rung 53
LD H185.12  ; 16ST_STEP 12
AND W123.05  ; 16ST_HOME POSITION
OR 4855.15  ; 16ST_CYCLE COMPLETE
LDNOT Bearing_Exchange_Edit
AND H185.07  ; 16ST_STEP 07
AND 2030.03  ; DROP GUARD FORWARD END
LD H0.10  ; LANE 1 CONFIRMATION THE OPERATION
OR W1.02  ; CYCLE STOP
ANDLD
ORLD
AND 4855.00  ; 16ST_CYCLE RUNNING
OUT 4855.15  ; 16ST_CYCLE COMPLETE
; rung 54: INDIV.
LD 1208.03  ; INDIVIDUAL OPERATION CIRCUIT EFFECTIVE
JMP(004) #16
; rung 55
LD W1.05  ; OPERATION INDIVIDUAL SELECT
AND 2090.07  ; MASTER ON CONFIRM
ANDNOT 4853.01  ; 16ST_1CY RUN
IL(002)
; rung 56
LD W70.00  ; POSITIONING 1 BACKWARD
AND 3800.00  ; SURE PUSH BUTTON SWITCH ON
LD 4853.03  ; 16ST_UNIT HOME POSITION PB
AND T1863  ; NO EXCHANGE CONTAINER
ORLD
AND 2030.01  ; LIFTER UPWARD END
OUT 4890.00  ; POSITIONING 1 BACKWARD

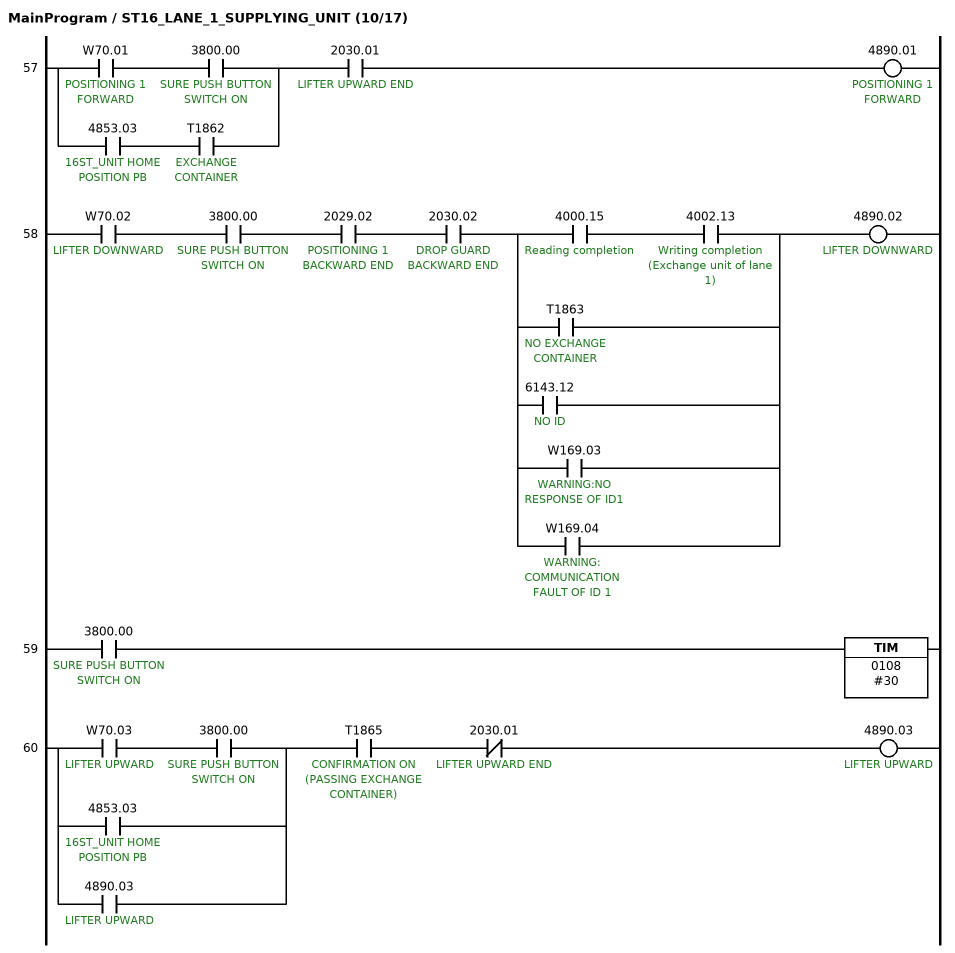
; rung 57
LD W70.01  ; POSITIONING 1 FORWARD
AND 3800.00  ; SURE PUSH BUTTON SWITCH ON
LD 4853.03  ; 16ST_UNIT HOME POSITION PB
AND T1862  ; EXCHANGE CONTAINER
ORLD
AND 2030.01  ; LIFTER UPWARD END
OUT 4890.01  ; POSITIONING 1 FORWARD
; rung 58
LD W70.02  ; LIFTER DOWNWARD
AND 3800.00  ; SURE PUSH BUTTON SWITCH ON
AND 2029.02  ; POSITIONING 1 BACKWARD END
AND 2030.02  ; DROP GUARD BACKWARD END
LD 4000.15  ; Reading completion
AND 4002.13  ; Writing completion (Exchange unit of lane 1)
OR T1863  ; NO EXCHANGE CONTAINER
OR 6143.12  ; NO ID
OR W169.03  ; WARNING:NO RESPONSE OF ID1
OR W169.04  ; WARNING:COMMUNICATION FAULT OF ID 1
ANDLD
OUT 4890.02  ; LIFTER DOWNWARD
; rung 59
LD 3800.00  ; SURE PUSH BUTTON SWITCH ON
TIM 0108 #30
; rung 60
LD W70.03  ; LIFTER UPWARD
AND 3800.00  ; SURE PUSH BUTTON SWITCH ON
OR 4853.03  ; 16ST_UNIT HOME POSITION PB
OR 4890.03  ; LIFTER UPWARD
AND T1865  ; CONFIRMATION ON (PASSING EXCHANGE CONTAINER)
ANDNOT 2030.01  ; LIFTER UPWARD END
OUT 4890.03  ; LIFTER UPWARD

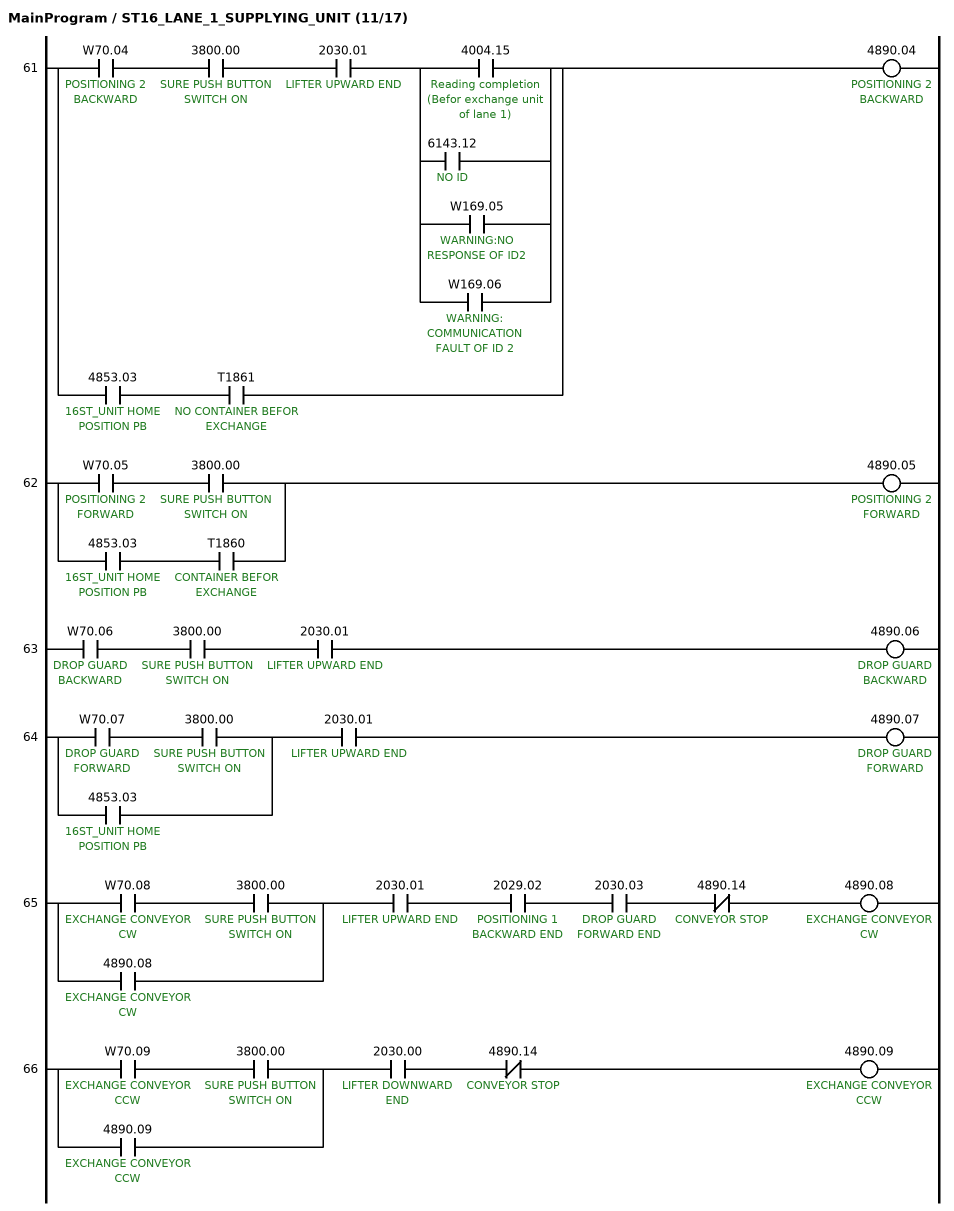
; rung 61
LD W70.04  ; POSITIONING 2 BACKWARD
AND 3800.00  ; SURE PUSH BUTTON SWITCH ON
AND 2030.01  ; LIFTER UPWARD END
LD 4004.15  ; Reading completion (Befor exchange unit of lane 1)
OR 6143.12  ; NO ID
OR W169.05  ; WARNING:NO RESPONSE OF ID2
OR W169.06  ; WARNING:COMMUNICATION FAULT OF ID 2
ANDLD
LD 4853.03  ; 16ST_UNIT HOME POSITION PB
AND T1861  ; NO CONTAINER BEFOR EXCHANGE
ORLD
OUT 4890.04  ; POSITIONING 2 BACKWARD
; rung 62
LD W70.05  ; POSITIONING 2 FORWARD
AND 3800.00  ; SURE PUSH BUTTON SWITCH ON
LD 4853.03  ; 16ST_UNIT HOME POSITION PB
AND T1860  ; CONTAINER BEFOR EXCHANGE
ORLD
OUT 4890.05  ; POSITIONING 2 FORWARD
; rung 63
LD W70.06  ; DROP GUARD BACKWARD
AND 3800.00  ; SURE PUSH BUTTON SWITCH ON
AND 2030.01  ; LIFTER UPWARD END
OUT 4890.06  ; DROP GUARD BACKWARD
; rung 64
LD W70.07  ; DROP GUARD FORWARD
AND 3800.00  ; SURE PUSH BUTTON SWITCH ON
OR 4853.03  ; 16ST_UNIT HOME POSITION PB
AND 2030.01  ; LIFTER UPWARD END
OUT 4890.07  ; DROP GUARD FORWARD
; rung 65
LD W70.08  ; EXCHANGE CONVEYOR CW
AND 3800.00  ; SURE PUSH BUTTON SWITCH ON
OR 4890.08  ; EXCHANGE CONVEYOR CW
AND 2030.01  ; LIFTER UPWARD END
AND 2029.02  ; POSITIONING 1 BACKWARD END
AND 2030.03  ; DROP GUARD FORWARD END
ANDNOT 4890.14  ; CONVEYOR STOP
OUT 4890.08  ; EXCHANGE CONVEYOR CW
; rung 66
LD W70.09  ; EXCHANGE CONVEYOR CCW
AND 3800.00  ; SURE PUSH BUTTON SWITCH ON
OR 4890.09  ; EXCHANGE CONVEYOR CCW
AND 2030.00  ; LIFTER DOWNWARD END
ANDNOT 4890.14  ; CONVEYOR STOP
OUT 4890.09  ; EXCHANGE CONVEYOR CCW

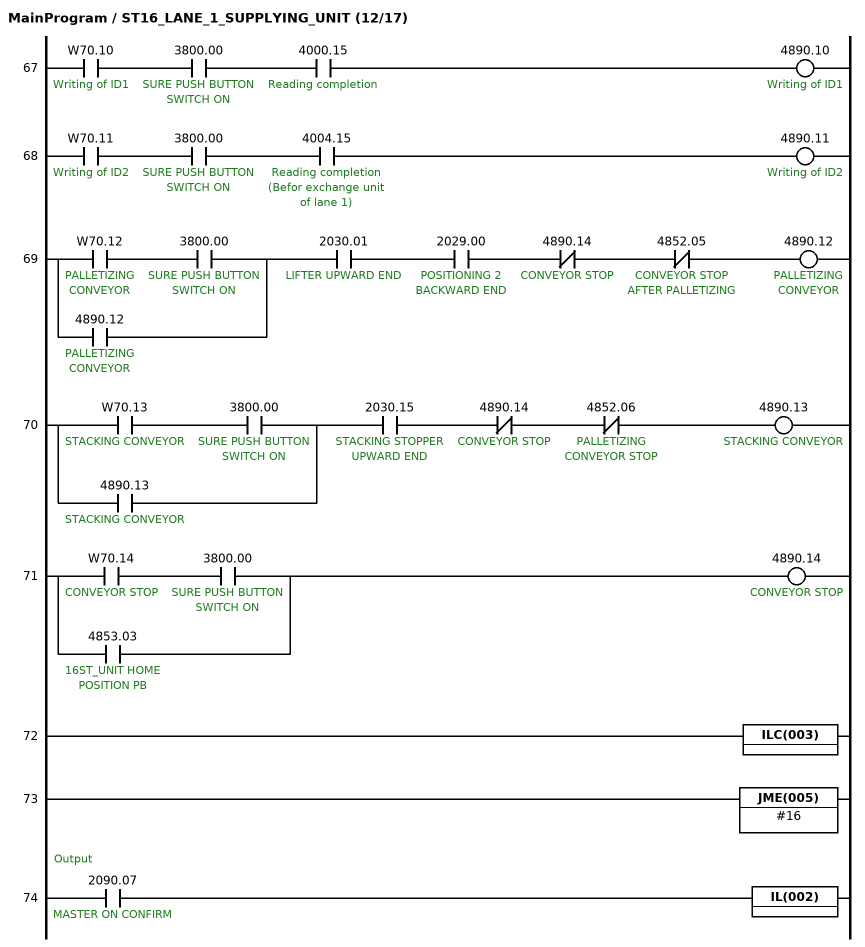
; rung 67
LD W70.10  ; Writing of ID1
AND 3800.00  ; SURE PUSH BUTTON SWITCH ON
AND 4000.15  ; Reading completion
OUT 4890.10  ; Writing of ID1
; rung 68
LD W70.11  ; Writing of ID2
AND 3800.00  ; SURE PUSH BUTTON SWITCH ON
AND 4004.15  ; Reading completion (Befor exchange unit of lane 1)
OUT 4890.11  ; Writing of ID2
; rung 69
LD W70.12  ; PALLETIZING CONVEYOR
AND 3800.00  ; SURE PUSH BUTTON SWITCH ON
OR 4890.12  ; PALLETIZING CONVEYOR
AND 2030.01  ; LIFTER UPWARD END
AND 2029.00  ; POSITIONING 2 BACKWARD END
ANDNOT 4890.14  ; CONVEYOR STOP
ANDNOT 4852.05  ; CONVEYOR STOP AFTER PALLETIZING
OUT 4890.12  ; PALLETIZING CONVEYOR
; rung 70
LD W70.13  ; STACKING CONVEYOR
AND 3800.00  ; SURE PUSH BUTTON SWITCH ON
OR 4890.13  ; STACKING CONVEYOR
AND 2030.15  ; STACKING STOPPER UPWARD END
ANDNOT 4890.14  ; CONVEYOR STOP
ANDNOT 4852.06  ; PALLETIZING CONVEYOR STOP
OUT 4890.13  ; STACKING CONVEYOR
; rung 71
LD W70.14  ; CONVEYOR STOP
AND 3800.00  ; SURE PUSH BUTTON SWITCH ON
OR 4853.03  ; 16ST_UNIT HOME POSITION PB
OUT 4890.14  ; CONVEYOR STOP
; rung 72
ILC(003)
; rung 73
JME(005) #16
; rung 74: Output
LD 2090.07  ; MASTER ON CONFIRM
IL(002)

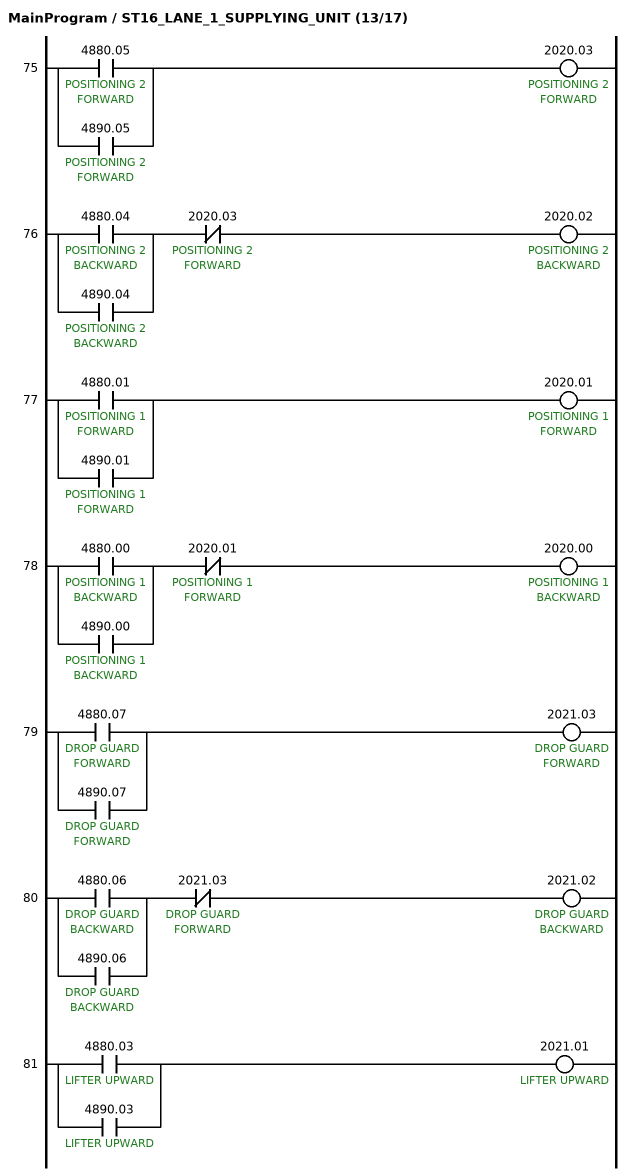
; rung 75
LD 4880.05  ; POSITIONING 2 FORWARD
OR 4890.05  ; POSITIONING 2 FORWARD
OUT 2020.03  ; POSITIONING 2 FORWARD
; rung 76
LD 4880.04  ; POSITIONING 2 BACKWARD
OR 4890.04  ; POSITIONING 2 BACKWARD
ANDNOT 2020.03  ; POSITIONING 2 FORWARD
OUT 2020.02  ; POSITIONING 2 BACKWARD
; rung 77
LD 4880.01  ; POSITIONING 1 FORWARD
OR 4890.01  ; POSITIONING 1 FORWARD
OUT 2020.01  ; POSITIONING 1 FORWARD
; rung 78
LD 4880.00  ; POSITIONING 1 BACKWARD
OR 4890.00  ; POSITIONING 1 BACKWARD
ANDNOT 2020.01  ; POSITIONING 1 FORWARD
OUT 2020.00  ; POSITIONING 1 BACKWARD
; rung 79
LD 4880.07  ; DROP GUARD FORWARD
OR 4890.07  ; DROP GUARD FORWARD
OUT 2021.03  ; DROP GUARD FORWARD
; rung 80
LD 4880.06  ; DROP GUARD BACKWARD
OR 4890.06  ; DROP GUARD BACKWARD
ANDNOT 2021.03  ; DROP GUARD FORWARD
OUT 2021.02  ; DROP GUARD BACKWARD
; rung 81
LD 4880.03  ; LIFTER UPWARD
OR 4890.03  ; LIFTER UPWARD
OUT 2021.01  ; LIFTER UPWARD

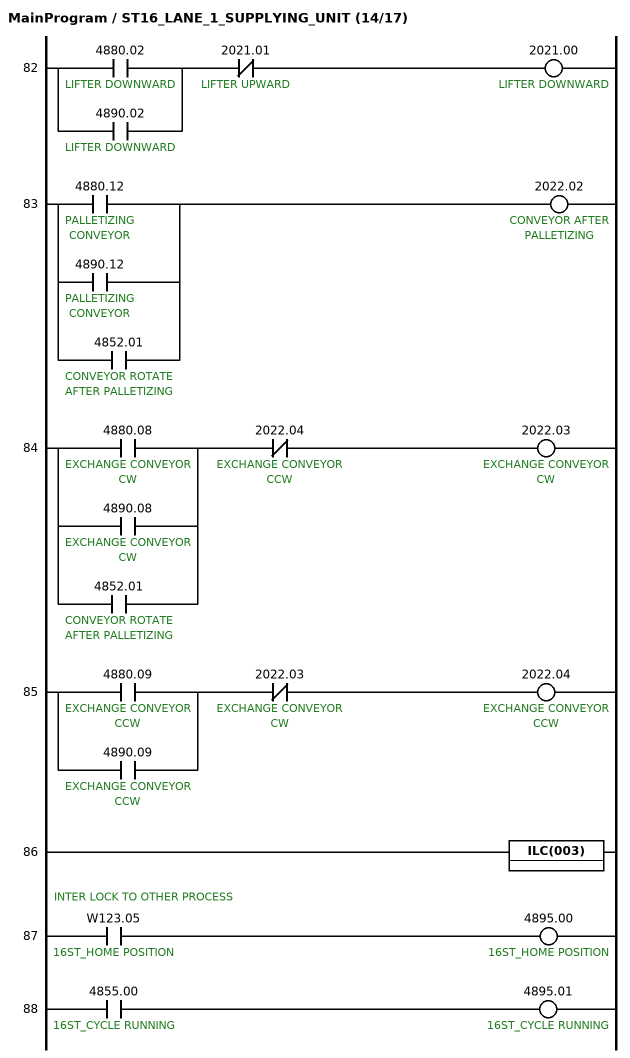
; rung 82
LD 4880.02  ; LIFTER DOWNWARD
OR 4890.02  ; LIFTER DOWNWARD
ANDNOT 2021.01  ; LIFTER UPWARD
OUT 2021.00  ; LIFTER DOWNWARD
; rung 83
LD 4880.12  ; PALLETIZING CONVEYOR
OR 4890.12  ; PALLETIZING CONVEYOR
OR 4852.01  ; CONVEYOR ROTATE AFTER PALLETIZING
OUT 2022.02  ; CONVEYOR AFTER PALLETIZING
; rung 84
LD 4880.08  ; EXCHANGE CONVEYOR CW
OR 4890.08  ; EXCHANGE CONVEYOR CW
OR 4852.01  ; CONVEYOR ROTATE AFTER PALLETIZING
ANDNOT 2022.04  ; EXCHANGE CONVEYOR CCW
OUT 2022.03  ; EXCHANGE CONVEYOR CW
; rung 85
LD 4880.09  ; EXCHANGE CONVEYOR CCW
OR 4890.09  ; EXCHANGE CONVEYOR CCW
ANDNOT 2022.03  ; EXCHANGE CONVEYOR CW
OUT 2022.04  ; EXCHANGE CONVEYOR CCW
; rung 86
ILC(003)
; rung 87: INTER LOCK TO OTHER PROCESS
LD W123.05  ; 16ST_HOME POSITION
OUT 4895.00  ; 16ST_HOME POSITION
; rung 88
LD 4855.00  ; 16ST_CYCLE RUNNING
OUT 4895.01  ; 16ST_CYCLE RUNNING

